LIN {X 0,Y 520.02,Z 1005.962,A -85,B 0,C 180,E1 24758.515,E2 24758.515} C_VEL
LIN {X 0,Y 519.949,Z 1010.979,A -85,B 0,C 180,E1 24756.515,E2 24756.515} C_VEL
LIN {X 0,Y 519.92,Z 1015.106,A -85,B 0,C 180,E1 24754.191,E2 24754.191} C_VEL
LIN {X 0,Y 519.914,Z 1017.318,A -85,B 0,C 180,E1 24751.984,E2 24751.984} C_VEL
LIN {X 0,Y 519.902,Z 1017.94,A -85,B 0,C 180,E1 24749.67,E2 24749.67} C_VEL
LIN {X 0,Y 519.907,Z 1016.99,A -85,B 0,C 180,E1 24747.576,E2 24747.576} C_VEL
LIN {X 0,Y 519.922,Z 1014.322,A -85,B 0,C 180,E1 24745.257,E2 24745.257} C_VEL
LIN {X 0,Y 519.954,Z 1010.226,A -85,B 0,C 180,E1 24743.153,E2 24743.153} C_VEL
LIN {X 0,Y 520.031,Z 1004.711,A -85,B 0,C 180,E1 24741.041,E2 24741.041} C_VEL
LIN {X 0,Y 520.195,Z 996.956,A -85,B 0,C 180,E1 24738.807,E2 24738.807} C_VEL
LIN {X 0,Y 520.466,Z 988.312,A -85,B 0,C 180,E1 24736.785,E2 24736.785} C_VEL
LIN {X 0,Y 520.856,Z 977.732,A -85,B 0,C 180,E1 24734.753,E2 24734.753} C_VEL
LIN {X 0,Y 521.388,Z 965.862,A -85,B 0,C 180,E1 24732.824,E2 24732.824} C_VEL
LIN {X 0,Y 522.046,Z 952.484,A -85,B 0,C 180,E1 24730.999,E2 24730.999} C_VEL
LIN {X 0,Y 522.795,Z 938.835,A -85,B 0,C 180,E1 24729.397,E2 24729.397} C_VEL
LIN {X 0,Y 523.77,Z 921.534,A -85,B 0,C 180,E1 24727.674,E2 24727.674} C_VEL
LIN {X 0,Y 524.742,Z 904.295,A -85,B 0,C 180,E1 24726.235,E2 24726.235} C_VEL
LIN {X 0,Y 525.694,Z 885.972,A -85,B 0,C 180,E1 24724.964,E2 24724.964} C_VEL
LIN {X 0,Y 526.661,Z 866.688,A -85,B 0,C 180,E1 24723.868,E2 24723.868} C_VEL
LIN {X 0,Y 527.517,Z 847.072,A -85,B 0,C 180,E1 24722.979,E2 24722.979} C_VEL
LIN {X 0,Y 528.202,Z 826.709,A -85,B 0,C 180,E1 24722.278,E2 24722.278} C_VEL
LIN {X 0,Y 528.779,Z 805.763,A -85,B 0,C 180,E1 24721.772,E2 24721.772} C_VEL
LIN {X 0,Y 529.175,Z 772.046,A -85,B 0,C 180,E1 24721.252,E2 24721.252} C_VEL
LIN {X 0,Y 534.131,Z 754.98,A -85,B 0,C 180,E1 24720.384,E2 24720.384} C_VEL
LIN {X 0,Y 537.725,Z 746.024,A -85,B 0,C 180,E1 24719.988,E2 24719.988} C_VEL
LIN {X 0,Y 541.751,Z 735.129,A -85,B 0,C 180,E1 24719.5,E2 24719.5} C_VEL
LIN {X 0,Y 548.246,Z 721.737,A -85,B 0,C 180,E1 24719.05,E2 24719.05} C_VEL
LIN {X 0,Y 556.194,Z 706.531,A -85,B 0,C 180,E1 24718.739,E2 24718.739} C_VEL
LIN {X 0,Y 561.276,Z 695.809,A -85,B 0,C 180,E1 24718.597,E2 24718.597} C_VEL
LIN {X 0,Y 565.411,Z 684.381,A -85,B 0,C 180,E1 24718.275,E2 24718.275} C_VEL
LIN {X 0,Y 572.184,Z 665.163,A -85,B 0,C 180,E1 24717.972,E2 24717.972} C_VEL
LIN {X 0,Y 577.855,Z 644.455,A -85,B 0,C 180,E1 24717.756,E2 24717.756} C_VEL
LIN {X 0,Y 581.468,Z 624.036,A -85,B 0,C 180,E1 24717.559,E2 24717.559} C_VEL
LIN {X 0,Y 581.827,Z 621.745,A -85,B 0,C 180,E1 24717.519,E2 24717.519} C_VEL
LIN {X 0,Y 583.33,Z 625.442,A -85,B 0,C 180,E1 24716.971,E2 24716.971} C_VEL
LIN {X 0,Y 583.255,Z 628.304,A -85,B 0,C 180,E1 24716.379,E2 24716.379} C_VEL
LIN {X 0,Y 581.69,Z 630.179,A -85,B 0,C 180,E1 24715.769,E2 24715.769} C_VEL
LIN {X 0,Y 578.618,Z 631.026,A -85,B 0,C 180,E1 24715.165,E2 24715.165} C_VEL
LIN {X 0,Y 574.8,Z 630.645,A -85,B 0,C 180,E1 24714.668,E2 24714.668} C_VEL
LIN {X 0,Y 568.857,Z 628.613,A -85,B 0,C 180,E1 24714.123,E2 24714.123} C_VEL
LIN {X 0,Y 560.136,Z 623.948,A -85,B 0,C 180,E1 24713.271,E2 24713.271} C_VEL
LIN {X 0,Y 552.133,Z 617.574,A -85,B 0,C 180,E1 24712.313,E2 24712.313} C_VEL
LIN {X 0,Y 545.581,Z 609.876,A -85,B 0,C 180,E1 24711.323,E2 24711.323} C_VEL
LIN {X 0,Y 540.263,Z 600.41,A -85,B 0,C 180,E1 24710.26,E2 24710.26} C_VEL
LIN {X 0,Y 536.466,Z 589.095,A -85,B 0,C 180,E1 24709.143,E2 24709.143} C_VEL
LIN {X 0,Y 534.195,Z 576.156,A -85,B 0,C 180,E1 24707.993,E2 24707.993} C_VEL
LIN {X 0,Y 533.452,Z 558.89,A -85,B 0,C 180,E1 24706.613,E2 24706.613} C_VEL
LIN {X 0,Y 535.809,Z 510.668,A -85,B 0,C 180,E1 24702.989,E2 24702.989} C_VEL
LIN {X 0,Y 537.167,Z 485.07,A -85,B 0,C 180,E1 24701.005,E2 24701.005} C_VEL
LIN {X 0,Y 528.374,Z 467.062,A -85,B 0,C 180,E1 24698.504,E2 24698.504} C_VEL
LIN {X 0,Y 523.968,Z 458.341,A -85,B 0,C 180,E1 24697.222,E2 24697.222} C_VEL
LIN {X 0,Y 521.991,Z 454.315,A -85,B 0,C 180,E1 24696.624,E2 24696.624} C_VEL
LIN {X 0,Y 520.59,Z 450.764,A -85,B 0,C 180,E1 24696.131,E2 24696.131} C_VEL
LIN {X 0,Y 520.581,Z 450.636,A -85,B 0,C 180,E1 24692.729,E2 24692.729} C_VEL
LIN {X 0,Y 520.553,Z 450.643,A -85,B 0,C 180,E1 24689.306,E2 24689.306} C_VEL
LIN {X 0,Y 520.585,Z 450.64,A -85,B 0,C 180,E1 24685.848,E2 24685.848} C_VEL
LIN {X 0,Y 520.561,Z 450.642,A -85,B 0,C 180,E1 24682.471,E2 24682.471} C_VEL
LIN {X 0,Y 520.537,Z 450.644,A -85,B 0,C 180,E1 24678.942,E2 24678.942} C_VEL
LIN {X 0,Y 520.586,Z 450.638,A -85,B 0,C 180,E1 24675.598,E2 24675.598} C_VEL
LIN {X 0,Y 520.533,Z 450.645,A -85,B 0,C 180,E1 24672.198,E2 24672.198} C_VEL
LIN {X 0,Y 520.562,Z 450.641,A -85,B 0,C 180,E1 24668.616,E2 24668.616} C_VEL
LIN {X 0,Y 520.585,Z 450.639,A -85,B 0,C 180,E1 24665.179,E2 24665.179} C_VEL
LIN {X 0,Y 520.563,Z 450.644,A -85,B 0,C 180,E1 24661.651,E2 24661.651} C_VEL
LIN {X 0,Y 520.583,Z 450.641,A -85,B 0,C 180,E1 24658.239,E2 24658.239} C_VEL
LIN {X 0,Y 520.573,Z 450.644,A -85,B 0,C 180,E1 24654.821,E2 24654.821} C_VEL
LIN {X 0,Y 520.584,Z 450.635,A -85,B 0,C 180,E1 24651.384,E2 24651.384} C_VEL
LIN {X 0,Y 520.559,Z 450.637,A -85,B 0,C 180,E1 24647.915,E2 24647.915} C_VEL
LIN {X 0,Y 520.582,Z 450.639,A -85,B 0,C 180,E1 24644.401,E2 24644.401} C_VEL
LIN {X 0,Y 520.565,Z 450.638,A -85,B 0,C 180,E1 24640.942,E2 24640.942} C_VEL
LIN {X 0,Y 520.533,Z 450.636,A -85,B 0,C 180,E1 24637.408,E2 24637.408} C_VEL
LIN {X 0,Y 520.584,Z 450.636,A -85,B 0,C 180,E1 24634.008,E2 24634.008} C_VEL
LIN {X 0,Y 520.541,Z 450.644,A -85,B 0,C 180,E1 24630.672,E2 24630.672} C_VEL
LIN {X 0,Y 520.557,Z 450.643,A -85,B 0,C 180,E1 24627.204,E2 24627.204} C_VEL
LIN {X 0,Y 520.586,Z 450.639,A -85,B 0,C 180,E1 24623.732,E2 24623.732} C_VEL
LIN {X 0,Y 520.556,Z 450.645,A -85,B 0,C 180,E1 24620.237,E2 24620.237} C_VEL
LIN {X 0,Y 520.586,Z 450.64,A -85,B 0,C 180,E1 24617.852,E2 24617.852} C_VEL
LIN {X 0,Y 519.595,Z 450.764,A -85,B 0,C 180,E1 24617.004,E2 24617.004} C_VEL
LIN {X 0,Y 513.124,Z 451.571,A -85,B 0,C 180,E1 24614.622,E2 24614.622} C_VEL
LIN {X 0,Y 512.608,Z 451.631,A -85,B 0,C 180,E1 24614.001,E2 24614.001} C_VEL
LIN {X 0,Y 512.622,Z 451.634,A -85,B 0,C 180,E1 24610.475,E2 24610.475} C_VEL
LIN {X 0,Y 512.655,Z 451.706,A -85,B 0,C 180,E1 24607.253,E2 24607.253} C_VEL
LIN {X 0,Y 522.069,Z 477.016,A -85,B 0,C 180,E1 24604.288,E2 24604.288} C_VEL
LIN {X 0,Y 521.564,Z 496.747,A -85,B 0,C 180,E1 24602.718,E2 24602.718} C_VEL
LIN {X 0,Y 524.472,Z 512.948,A -85,B 0,C 180,E1 24602.253,E2 24602.253} C_VEL
LIN {X 0,Y 521.733,Z 755.843,A -85,B 0,C 180,E1 24598.599,E2 24598.599} C_VEL
LIN {X 0,Y 521.118,Z 776.945,A -85,B 0,C 180,E1 24598.086,E2 24598.086} C_VEL
LIN {X 0,Y 520.343,Z 797.387,A -85,B 0,C 180,E1 24597.369,E2 24597.369} C_VEL
LIN {X 0,Y 519.455,Z 815.917,A -85,B 0,C 180,E1 24596.522,E2 24596.522} C_VEL
LIN {X 0,Y 518.399,Z 835.331,A -85,B 0,C 180,E1 24595.413,E2 24595.413} C_VEL
LIN {X 0,Y 517.335,Z 853.73,A -85,B 0,C 180,E1 24594.127,E2 24594.127} C_VEL
LIN {X 0,Y 516.225,Z 871.52,A -85,B 0,C 180,E1 24592.628,E2 24592.628} C_VEL
LIN {X 0,Y 515.211,Z 887.582,A -85,B 0,C 180,E1 24591.018,E2 24591.018} C_VEL
LIN {X 0,Y 514.336,Z 902.16,A -85,B 0,C 180,E1 24589.297,E2 24589.297} C_VEL
LIN {X 0,Y 513.544,Z 916.286,A -85,B 0,C 180,E1 24587.33,E2 24587.33} C_VEL
LIN {X 0,Y 512.924,Z 928.972,A -85,B 0,C 180,E1 24585.221,E2 24585.221} C_VEL
LIN {X 0,Y 512.488,Z 939.658,A -85,B 0,C 180,E1 24583.08,E2 24583.08} C_VEL
LIN {X 0,Y 512.196,Z 948.513,A -85,B 0,C 180,E1 24580.914,E2 24580.914} C_VEL
LIN {X 0,Y 512.04,Z 955.576,A -85,B 0,C 180,E1 24578.76,E2 24578.76} C_VEL
LIN {X 0,Y 511.954,Z 961.153,A -85,B 0,C 180,E1 24576.504,E2 24576.504} C_VEL
LIN {X 0,Y 511.921,Z 965.02,A -85,B 0,C 180,E1 24574.256,E2 24574.256} C_VEL
LIN {X 0,Y 511.912,Z 967.346,A -85,B 0,C 180,E1 24571.902,E2 24571.902} C_VEL
LIN {X 0,Y 511.903,Z 967.949,A -85,B 0,C 180,E1 24569.664,E2 24569.664} C_VEL
LIN {X 0,Y 511.906,Z 966.99,A -85,B 0,C 180,E1 24567.425,E2 24567.425} C_VEL
LIN {X 0,Y 511.924,Z 964.355,A -85,B 0,C 180,E1 24565.182,E2 24565.182} C_VEL
LIN {X 0,Y 511.958,Z 960.09,A -85,B 0,C 180,E1 24562.932,E2 24562.932} C_VEL
LIN {X 0,Y 512.054,Z 954.108,A -85,B 0,C 180,E1 24560.672,E2 24560.672} C_VEL
LIN {X 0,Y 512.254,Z 946.567,A -85,B 0,C 180,E1 24558.478,E2 24558.478} C_VEL
LIN {X 0,Y 512.578,Z 937.474,A -85,B 0,C 180,E1 24556.347,E2 24556.347} C_VEL
LIN {X 0,Y 513.066,Z 926.091,A -85,B 0,C 180,E1 24554.167,E2 24554.167} C_VEL
LIN {X 0,Y 513.736,Z 913.04,A -85,B 0,C 180,E1 24552.09,E2 24552.09} C_VEL
LIN {X 0,Y 514.521,Z 899.191,A -85,B 0,C 180,E1 24550.236,E2 24550.236} C_VEL
LIN {X 0,Y 515.417,Z 884.365,A -85,B 0,C 180,E1 24548.55,E2 24548.55} C_VEL
LIN {X 0,Y 516.418,Z 868.089,A -85,B 0,C 180,E1 24546.976,E2 24546.976} C_VEL
LIN {X 0,Y 517.483,Z 850.915,A -85,B 0,C 180,E1 24545.576,E2 24545.576} C_VEL
LIN {X 0,Y 518.537,Z 832.917,A -85,B 0,C 180,E1 24544.348,E2 24544.348} C_VEL
LIN {X 0,Y 519.552,Z 814.203,A -85,B 0,C 180,E1 24543.297,E2 24543.297} C_VEL
LIN {X 0,Y 520.482,Z 794.444,A -85,B 0,C 180,E1 24542.421,E2 24542.421} C_VEL
LIN {X 0,Y 521.208,Z 774.575,A -85,B 0,C 180,E1 24541.755,E2 24541.755} C_VEL
LIN {X 0,Y 521.766,Z 754.007,A -85,B 0,C 180,E1 24541.277,E2 24541.277} C_VEL
LIN {X 0,Y 524.313,Z 517.721,A -85,B 0,C 180,E1 24537.722,E2 24537.722} C_VEL
LIN {X 0,Y 519.038,Z 498.46,A -85,B 0,C 180,E1 24537.028,E2 24537.028} C_VEL
LIN {X 0,Y 519.95,Z 475.219,A -85,B 0,C 180,E1 24534.157,E2 24534.157} C_VEL
LIN {X 0,Y 514.832,Z 458.731,A -85,B 0,C 180,E1 24531.575,E2 24531.575} C_VEL
LIN {X 0,Y 512.627,Z 451.637,A -85,B 0,C 180,E1 24530.417,E2 24530.417} C_VEL
LIN {X 0,Y 512.646,Z 451.628,A -85,B 0,C 180,E1 24526.949,E2 24526.949} C_VEL
LIN {X 0,Y 512.633,Z 451.628,A -85,B 0,C 180,E1 24523.483,E2 24523.483} C_VEL
LIN {X 0,Y 512.63,Z 451.628,A -85,B 0,C 180,E1 24519.919,E2 24519.919} C_VEL
LIN {X 0,Y 512.638,Z 451.63,A -85,B 0,C 180,E1 24516.504,E2 24516.504} C_VEL
LIN {X 0,Y 512.638,Z 451.637,A -85,B 0,C 180,E1 24512.968,E2 24512.968} C_VEL
LIN {X 0,Y 512.667,Z 451.773,A -85,B 0,C 180,E1 24512.038,E2 24512.038} C_VEL
LIN {X 0,Y 520.423,Z 474.252,A -85,B 0,C 180,E1 24509.053,E2 24509.053} C_VEL
LIN {X 0,Y 521.005,Z 476.298,A -85,B 0,C 180,E1 24508.796,E2 24508.796} C_VEL
LIN {X 0,Y 519.755,Z 507.875,A -85,B 0,C 180,E1 24505.648,E2 24505.648} C_VEL
LIN {X 0,Y 518.449,Z 542.34,A -85,B 0,C 180,E1 24502.269,E2 24502.269} C_VEL
LIN {X 0,Y 517.128,Z 577.872,A -85,B 0,C 180,E1 24498.838,E2 24498.838} C_VEL
LIN {X 0,Y 516.275,Z 609.248,A -85,B 0,C 180,E1 24495.884,E2 24495.884} C_VEL
LIN {X 0,Y 516.883,Z 614.725,A -85,B 0,C 180,E1 24495.767,E2 24495.767} C_VEL
LIN {X 0,Y 515.399,Z 751.101,A -85,B 0,C 180,E1 24493.597,E2 24493.597} C_VEL
LIN {X 0,Y 515.196,Z 767.868,A -85,B 0,C 180,E1 24493.11,E2 24493.11} C_VEL
LIN {X 0,Y 514.884,Z 783.198,A -85,B 0,C 180,E1 24492.448,E2 24492.448} C_VEL
LIN {X 0,Y 514.483,Z 798.649,A -85,B 0,C 180,E1 24491.547,E2 24491.547} C_VEL
LIN {X 0,Y 514.057,Z 812.03,A -85,B 0,C 180,E1 24490.535,E2 24490.535} C_VEL
LIN {X 0,Y 513.602,Z 825.042,A -85,B 0,C 180,E1 24489.299,E2 24489.299} C_VEL
LIN {X 0,Y 513.201,Z 836.355,A -85,B 0,C 180,E1 24487.951,E2 24487.951} C_VEL
LIN {X 0,Y 512.843,Z 846.858,A -85,B 0,C 180,E1 24486.381,E2 24486.381} C_VEL
LIN {X 0,Y 512.595,Z 855.085,A -85,B 0,C 180,E1 24484.812,E2 24484.812} C_VEL
LIN {X 0,Y 512.416,Z 861.858,A -85,B 0,C 180,E1 24483.132,E2 24483.132} C_VEL
LIN {X 0,Y 512.306,Z 866.86,A -85,B 0,C 180,E1 24481.454,E2 24481.454} C_VEL
LIN {X 0,Y 512.257,Z 870.497,A -85,B 0,C 180,E1 24479.553,E2 24479.553} C_VEL
LIN {X 0,Y 512.241,Z 872.22,A -85,B 0,C 180,E1 24477.763,E2 24477.763} C_VEL
LIN {X 0,Y 512.262,Z 872.167,A -85,B 0,C 180,E1 24475.859,E2 24475.859} C_VEL
LIN {X 0,Y 512.314,Z 870.441,A -85,B 0,C 180,E1 24474.063,E2 24474.063} C_VEL
LIN {X 0,Y 512.407,Z 866.934,A -85,B 0,C 180,E1 24472.262,E2 24472.262} C_VEL
LIN {X 0,Y 512.594,Z 861.578,A -85,B 0,C 180,E1 24470.456,E2 24470.456} C_VEL
LIN {X 0,Y 512.822,Z 854.415,A -85,B 0,C 180,E1 24468.731,E2 24468.731} C_VEL
LIN {X 0,Y 513.149,Z 846.02,A -85,B 0,C 180,E1 24467.166,E2 24467.166} C_VEL
LIN {X 0,Y 513.505,Z 836.727,A -85,B 0,C 180,E1 24465.798,E2 24465.798} C_VEL
LIN {X 0,Y 513.961,Z 825.126,A -85,B 0,C 180,E1 24464.427,E2 24464.427} C_VEL
LIN {X 0,Y 514.405,Z 812.983,A -85,B 0,C 180,E1 24463.282,E2 24463.282} C_VEL
LIN {X 0,Y 514.82,Z 799.097,A -85,B 0,C 180,E1 24462.247,E2 24462.247} C_VEL
LIN {X 0,Y 515.154,Z 785.148,A -85,B 0,C 180,E1 24461.44,E2 24461.44} C_VEL
LIN {X 0,Y 515.389,Z 769.335,A -85,B 0,C 180,E1 24460.773,E2 24460.773} C_VEL
LIN {X 0,Y 515.494,Z 753.566,A -85,B 0,C 180,E1 24460.325,E2 24460.325} C_VEL
LIN {X 0,Y 517.063,Z 653.13,A -85,B 0,C 180,E1 24458.571,E2 24458.571} C_VEL
LIN {X 0,Y 517.869,Z 619.502,A -85,B 0,C 180,E1 24457.943,E2 24457.943} C_VEL
LIN {X 0,Y 519.364,Z 614.58,A -85,B 0,C 180,E1 24457.531,E2 24457.531} C_VEL
LIN {X 0,Y 522.354,Z 579.387,A -85,B 0,C 180,E1 24453.758,E2 24453.758} C_VEL
LIN {X 0,Y 526.373,Z 547.133,A -85,B 0,C 180,E1 24450.091,E2 24450.091} C_VEL
LIN {X 0,Y 530.894,Z 521.985,A -85,B 0,C 180,E1 24447.024,E2 24447.024} C_VEL
LIN {X 0,Y 534.242,Z 508.14,A -85,B 0,C 180,E1 24445.193,E2 24445.193} C_VEL
LIN {X 0,Y 536.725,Z 498.815,A -85,B 0,C 180,E1 24443.769,E2 24443.769} C_VEL
LIN {X 0,Y 536.061,Z 495.319,A -85,B 0,C 180,E1 24442.417,E2 24442.417} C_VEL
LIN {X 0,Y 536.022,Z 493.334,A -85,B 0,C 180,E1 24441.189,E2 24441.189} C_VEL
LIN {X 0,Y 536.329,Z 493.269,A -85,B 0,C 180,E1 24439.832,E2 24439.832} C_VEL
LIN {X 0,Y 536.826,Z 494.261,A -85,B 0,C 180,E1 24439.049,E2 24439.049} C_VEL
LIN {X 0,Y 531.613,Z 507.135,A -85,B 0,C 180,E1 24437.66,E2 24437.66} C_VEL
LIN {X 0,Y 527.47,Z 522.779,A -85,B 0,C 180,E1 24436.16,E2 24436.16} C_VEL
LIN {X 0,Y 523.936,Z 544.359,A -85,B 0,C 180,E1 24434.304,E2 24434.304} C_VEL
LIN {X 0,Y 522.918,Z 563.007,A -85,B 0,C 180,E1 24432.75,E2 24432.75} C_VEL
LIN {X 0,Y 523.903,Z 578.013,A -85,B 0,C 180,E1 24431.472,E2 24431.472} C_VEL
LIN {X 0,Y 526.805,Z 591.429,A -85,B 0,C 180,E1 24430.272,E2 24430.272} C_VEL
LIN {X 0,Y 531.066,Z 602.392,A -85,B 0,C 180,E1 24429.243,E2 24429.243} C_VEL
LIN {X 0,Y 537.171,Z 612.519,A -85,B 0,C 180,E1 24428.235,E2 24428.235} C_VEL
LIN {X 0,Y 544.544,Z 621.028,A -85,B 0,C 180,E1 24427.341,E2 24427.341} C_VEL
LIN {X 0,Y 553.465,Z 628.474,A -85,B 0,C 180,E1 24426.495,E2 24426.495} C_VEL
LIN {X 0,Y 563.066,Z 634.265,A -85,B 0,C 180,E1 24425.756,E2 24425.756} C_VEL
LIN {X 0,Y 569.587,Z 637.069,A -85,B 0,C 180,E1 24425.288,E2 24425.288} C_VEL
LIN {X 0,Y 573.909,Z 638.04,A -85,B 0,C 180,E1 24424.851,E2 24424.851} C_VEL
LIN {X 0,Y 577.534,Z 637.952,A -85,B 0,C 180,E1 24424.33,E2 24424.33} C_VEL
LIN {X 0,Y 580.243,Z 636.66,A -85,B 0,C 180,E1 24423.702,E2 24423.702} C_VEL
LIN {X 0,Y 581.263,Z 634.732,A -85,B 0,C 180,E1 24423.118,E2 24423.118} C_VEL
LIN {X 0,Y 574.611,Z 654.779,A -85,B 0,C 180,E1 24422.941,E2 24422.941} C_VEL
LIN {X 0,Y 566.188,Z 674.796,A -85,B 0,C 180,E1 24422.656,E2 24422.656} C_VEL
LIN {X 0,Y 558.971,Z 690.695,A -85,B 0,C 180,E1 24422.273,E2 24422.273} C_VEL
LIN {X 0,Y 556.522,Z 696.659,A -85,B 0,C 180,E1 24422.067,E2 24422.067} C_VEL
LIN {X 0,Y 546.748,Z 712.537,A -85,B 0,C 180,E1 24421.714,E2 24421.714} C_VEL
LIN {X 0,Y 538.402,Z 726.619,A -85,B 0,C 180,E1 24421.207,E2 24421.207} C_VEL
LIN {X 0,Y 532.513,Z 739.169,A -85,B 0,C 180,E1 24420.65,E2 24420.65} C_VEL
LIN {X 0,Y 529.342,Z 747.906,A -85,B 0,C 180,E1 24420.225,E2 24420.225} C_VEL
LIN {X 0,Y 525.03,Z 759.145,A -85,B 0,C 180,E1 24419.68,E2 24419.68} C_VEL
LIN {X 0,Y 521.684,Z 771.68,A -85,B 0,C 180,E1 24419.052,E2 24419.052} C_VEL
LIN {X 0,Y 521.265,Z 808.1,A -85,B 0,C 180,E1 24418.499,E2 24418.499} C_VEL
LIN {X 0,Y 520.716,Z 830.208,A -85,B 0,C 180,E1 24417.958,E2 24417.958} C_VEL
LIN {X 0,Y 520.042,Z 850.995,A -85,B 0,C 180,E1 24417.232,E2 24417.232} C_VEL
LIN {X 0,Y 519.241,Z 869.965,A -85,B 0,C 180,E1 24416.351,E2 24416.351} C_VEL
LIN {X 0,Y 518.204,Z 888.718,A -85,B 0,C 180,E1 24415.241,E2 24415.241} C_VEL
LIN {X 0,Y 517.097,Z 907.27,A -85,B 0,C 180,E1 24413.891,E2 24413.891} C_VEL
LIN {X 0,Y 516.031,Z 924.658,A -85,B 0,C 180,E1 24412.38,E2 24412.38} C_VEL
LIN {X 0,Y 515.042,Z 940.356,A -85,B 0,C 180,E1 24410.751,E2 24410.751} C_VEL
LIN {X 0,Y 514.26,Z 953.384,A -85,B 0,C 180,E1 24409.183,E2 24409.183} C_VEL
LIN {X 0,Y 513.49,Z 967.318,A -85,B 0,C 180,E1 24407.216,E2 24407.216} C_VEL
LIN {X 0,Y 512.95,Z 978.366,A -85,B 0,C 180,E1 24405.373,E2 24405.373} C_VEL
LIN {X 0,Y 512.48,Z 989.843,A -85,B 0,C 180,E1 24403.081,E2 24403.081} C_VEL
LIN {X 0,Y 512.191,Z 998.694,A -85,B 0,C 180,E1 24400.914,E2 24400.914} C_VEL
LIN {X 0,Y 512.033,Z 1005.958,A -85,B 0,C 180,E1 24398.648,E2 24398.648} C_VEL
LIN {X 0,Y 511.955,Z 1010.977,A -85,B 0,C 180,E1 24396.617,E2 24396.617} C_VEL
LIN {X 0,Y 511.919,Z 1015.101,A -85,B 0,C 180,E1 24394.257,E2 24394.257} C_VEL
LIN {X 0,Y 511.914,Z 1017.314,A -85,B 0,C 180,E1 24392.015,E2 24392.015} C_VEL
LIN {X 0,Y 511.902,Z 1017.94,A -85,B 0,C 180,E1 24389.665,E2 24389.665} C_VEL
LIN {X 0,Y 511.907,Z 1016.985,A -85,B 0,C 180,E1 24387.538,E2 24387.538} C_VEL
LIN {X 0,Y 511.923,Z 1014.322,A -85,B 0,C 180,E1 24385.183,E2 24385.183} C_VEL
LIN {X 0,Y 511.957,Z 1010.224,A -85,B 0,C 180,E1 24383.046,E2 24383.046} C_VEL
LIN {X 0,Y 512.045,Z 1004.71,A -85,B 0,C 180,E1 24380.9,E2 24380.9} C_VEL
LIN {X 0,Y 512.223,Z 997.388,A -85,B 0,C 180,E1 24378.744,E2 24378.744} C_VEL
LIN {X 0,Y 512.519,Z 988.832,A -85,B 0,C 180,E1 24376.692,E2 24376.692} C_VEL
LIN {X 0,Y 512.979,Z 977.728,A -85,B 0,C 180,E1 24374.513,E2 24374.513} C_VEL
LIN {X 0,Y 513.58,Z 965.794,A -85,B 0,C 180,E1 24372.544,E2 24372.544} C_VEL
LIN {X 0,Y 514.31,Z 952.479,A -85,B 0,C 180,E1 24370.702,E2 24370.702} C_VEL
LIN {X 0,Y 515.136,Z 938.829,A -85,B 0,C 180,E1 24369.076,E2 24369.076} C_VEL
LIN {X 0,Y 516.22,Z 921.531,A -85,B 0,C 180,E1 24367.33,E2 24367.33} C_VEL
LIN {X 0,Y 517.306,Z 904.221,A -85,B 0,C 180,E1 24365.866,E2 24365.866} C_VEL
LIN {X 0,Y 518.352,Z 885.967,A -85,B 0,C 180,E1 24364.585,E2 24364.585} C_VEL
LIN {X 0,Y 519.339,Z 867.859,A -85,B 0,C 180,E1 24363.539,E2 24363.539} C_VEL
LIN {X 0,Y 520.181,Z 848.295,A -85,B 0,C 180,E1 24362.653,E2 24362.653} C_VEL
LIN {X 0,Y 520.884,Z 827.337,A -85,B 0,C 180,E1 24361.932,E2 24361.932} C_VEL
LIN {X 0,Y 521.509,Z 805.279,A -85,B 0,C 180,E1 24361.398,E2 24361.398} C_VEL
LIN {X 0,Y 522.015,Z 771.041,A -85,B 0,C 180,E1 24360.861,E2 24360.861} C_VEL
LIN {X 0,Y 527.015,Z 754.196,A -85,B 0,C 180,E1 24359.998,E2 24359.998} C_VEL
LIN {X 0,Y 530.862,Z 744.608,A -85,B 0,C 180,E1 24359.56,E2 24359.56} C_VEL
LIN {X 0,Y 535.34,Z 733.098,A -85,B 0,C 180,E1 24359.033,E2 24359.033} C_VEL
LIN {X 0,Y 542.601,Z 719.324,A -85,B 0,C 180,E1 24358.507,E2 24358.507} C_VEL
LIN {X 0,Y 552.028,Z 704.082,A -85,B 0,C 180,E1 24358.071,E2 24358.071} C_VEL
LIN {X 0,Y 556.94,Z 695.681,A -85,B 0,C 180,E1 24357.901,E2 24357.901} C_VEL
LIN {X 0,Y 562.319,Z 683.23,A -85,B 0,C 180,E1 24357.522,E2 24357.522} C_VEL
LIN {X 0,Y 570.851,Z 664.161,A -85,B 0,C 180,E1 24357.174,E2 24357.174} C_VEL
LIN {X 0,Y 578.175,Z 644.792,A -85,B 0,C 180,E1 24356.963,E2 24356.963} C_VEL
LIN {X 0,Y 581.311,Z 634.577,A -85,B 0,C 180,E1 24356.871,E2 24356.871} C_VEL
LIN {X 0,Y 580.248,Z 636.656,A -85,B 0,C 180,E1 24356.3,E2 24356.3} C_VEL
LIN {X 0,Y 578.071,Z 637.821,A -85,B 0,C 180,E1 24355.768,E2 24355.768} C_VEL
LIN {X 0,Y 574.538,Z 638.101,A -85,B 0,C 180,E1 24355.226,E2 24355.226} C_VEL
LIN {X 0,Y 570.275,Z 637.279,A -85,B 0,C 180,E1 24354.773,E2 24354.773} C_VEL
LIN {X 0,Y 560.456,Z 633.212,A -85,B 0,C 180,E1 24353.916,E2 24353.916} C_VEL
LIN {X 0,Y 551.304,Z 627.408,A -85,B 0,C 180,E1 24352.939,E2 24352.939} C_VEL
LIN {X 0,Y 543.628,Z 620.254,A -85,B 0,C 180,E1 24351.924,E2 24351.924} C_VEL
LIN {X 0,Y 537.412,Z 611.822,A -85,B 0,C 180,E1 24350.88,E2 24350.88} C_VEL
LIN {X 0,Y 532.658,Z 602.127,A -85,B 0,C 180,E1 24349.816,E2 24349.816} C_VEL
LIN {X 0,Y 529.071,Z 589.803,A -85,B 0,C 180,E1 24348.613,E2 24348.613} C_VEL
LIN {X 0,Y 527.134,Z 575.752,A -85,B 0,C 180,E1 24347.379,E2 24347.379} C_VEL
LIN {X 0,Y 526.882,Z 556.312,A -85,B 0,C 180,E1 24345.834,E2 24345.834} C_VEL
LIN {X 0,Y 529.293,Z 514.033,A -85,B 0,C 180,E1 24342.627,E2 24342.627} C_VEL
LIN {X 0,Y 530.745,Z 489.136,A -85,B 0,C 180,E1 24340.679,E2 24340.679} C_VEL
LIN {X 0,Y 522.147,Z 471.547,A -85,B 0,C 180,E1 24338.207,E2 24338.207} C_VEL
LIN {X 0,Y 515.983,Z 459.211,A -85,B 0,C 180,E1 24336.367,E2 24336.367} C_VEL
LIN {X 0,Y 514.262,Z 455.59,A -85,B 0,C 180,E1 24335.818,E2 24335.818} C_VEL
LIN {X 0,Y 512.684,Z 452.156,A -85,B 0,C 180,E1 24335.3,E2 24335.3} C_VEL
LIN {X 0,Y 512.605,Z 451.631,A -85,B 0,C 180,E1 24335.188,E2 24335.188} C_VEL
LIN {X 0,Y 512.644,Z 451.621,A -85,B 0,C 180,E1 24331.645,E2 24331.645} C_VEL
LIN {X 0,Y 512.617,Z 451.632,A -85,B 0,C 180,E1 24328.292,E2 24328.292} C_VEL
LIN {X 0,Y 512.641,Z 451.631,A -85,B 0,C 180,E1 24324.793,E2 24324.793} C_VEL
LIN {X 0,Y 512.639,Z 451.631,A -85,B 0,C 180,E1 24321.271,E2 24321.271} C_VEL
LIN {X 0,Y 512.651,Z 451.629,A -85,B 0,C 180,E1 24317.713,E2 24317.713} C_VEL
LIN {X 0,Y 512.622,Z 451.632,A -85,B 0,C 180,E1 24314.216,E2 24314.216} C_VEL
LIN {X 0,Y 512.597,Z 451.634,A -85,B 0,C 180,E1 24310.679,E2 24310.679} C_VEL
LIN {X 0,Y 512.651,Z 451.625,A -85,B 0,C 180,E1 24307.283,E2 24307.283} C_VEL
LIN {X 0,Y 512.594,Z 451.634,A -85,B 0,C 180,E1 24303.914,E2 24303.914} C_VEL
LIN {X 0,Y 512.622,Z 451.628,A -85,B 0,C 180,E1 24300.335,E2 24300.335} C_VEL
LIN {X 0,Y 512.645,Z 451.628,A -85,B 0,C 180,E1 24296.869,E2 24296.869} C_VEL
LIN {X 0,Y 512.631,Z 451.628,A -85,B 0,C 180,E1 24293.279,E2 24293.279} C_VEL
LIN {X 0,Y 512.641,Z 451.632,A -85,B 0,C 180,E1 24289.776,E2 24289.776} C_VEL
LIN {X 0,Y 512.627,Z 451.625,A -85,B 0,C 180,E1 24286.349,E2 24286.349} C_VEL
LIN {X 0,Y 512.645,Z 451.623,A -85,B 0,C 180,E1 24282.989,E2 24282.989} C_VEL
LIN {X 0,Y 512.618,Z 451.632,A -85,B 0,C 180,E1 24279.565,E2 24279.565} C_VEL
LIN {X 0,Y 512.637,Z 451.628,A -85,B 0,C 180,E1 24276.066,E2 24276.066} C_VEL
LIN {X 0,Y 512.627,Z 451.626,A -85,B 0,C 180,E1 24272.719,E2 24272.719} C_VEL
LIN {X 0,Y 512.594,Z 451.627,A -85,B 0,C 180,E1 24269.12,E2 24269.12} C_VEL
LIN {X 0,Y 512.644,Z 451.624,A -85,B 0,C 180,E1 24265.69,E2 24265.69} C_VEL
LIN {X 0,Y 512.602,Z 451.63,A -85,B 0,C 180,E1 24262.365,E2 24262.365} C_VEL
LIN {X 0,Y 512.617,Z 451.626,A -85,B 0,C 180,E1 24258.841,E2 24258.841} C_VEL
LIN {X 0,Y 512.651,Z 451.629,A -85,B 0,C 180,E1 24255.388,E2 24255.388} C_VEL
LIN {X 0,Y 512.608,Z 451.631,A -85,B 0,C 180,E1 24254.001,E2 24254.001} C_VEL
LIN {X 0,Y 511.64,Z 451.759,A -85,B 0,C 180,E1 24253.14,E2 24253.14} C_VEL
LIN {X 0,Y 505.215,Z 452.557,A -85,B 0,C 180,E1 24250.719,E2 24250.719} C_VEL
LIN {X 0,Y 504.704,Z 452.617,A -85,B 0,C 180,E1 24250.088,E2 24250.088} C_VEL
LIN {X 0,Y 504.702,Z 452.709,A -85,B 0,C 180,E1 24247.835,E2 24247.835} C_VEL
LIN {X 0,Y 513.665,Z 476.547,A -85,B 0,C 180,E1 24244.966,E2 24244.966} C_VEL
LIN {X 0,Y 515.013,Z 480.366,A -85,B 0,C 180,E1 24244.533,E2 24244.533} C_VEL
LIN {X 0,Y 514.614,Z 497.14,A -85,B 0,C 180,E1 24243.215,E2 24243.215} C_VEL
LIN {X 0,Y 517.714,Z 514.315,A -85,B 0,C 180,E1 24242.71,E2 24242.71} C_VEL
LIN {X 0,Y 514.722,Z 756.349,A -85,B 0,C 180,E1 24239.021,E2 24239.021} C_VEL
LIN {X 0,Y 514.073,Z 777.294,A -85,B 0,C 180,E1 24238.506,E2 24238.506} C_VEL
LIN {X 0,Y 513.25,Z 797.555,A -85,B 0,C 180,E1 24237.789,E2 24237.789} C_VEL
LIN {X 0,Y 512.279,Z 816.309,A -85,B 0,C 180,E1 24236.924,E2 24236.924} C_VEL
LIN {X 0,Y 511.192,Z 834.747,A -85,B 0,C 180,E1 24235.859,E2 24235.859} C_VEL
LIN {X 0,Y 509.955,Z 853.489,A -85,B 0,C 180,E1 24234.528,E2 24234.528} C_VEL
LIN {X 0,Y 508.683,Z 871.724,A -85,B 0,C 180,E1 24232.964,E2 24232.964} C_VEL
LIN {X 0,Y 507.598,Z 887.383,A -85,B 0,C 180,E1 24231.371,E2 24231.371} C_VEL
LIN {X 0,Y 506.619,Z 902.163,A -85,B 0,C 180,E1 24229.603,E2 24229.603} C_VEL
LIN {X 0,Y 505.742,Z 916.288,A -85,B 0,C 180,E1 24227.606,E2 24227.606} C_VEL
LIN {X 0,Y 505.059,Z 928.776,A -85,B 0,C 180,E1 24225.501,E2 24225.501} C_VEL
LIN {X 0,Y 504.573,Z 939.379,A -85,B 0,C 180,E1 24223.353,E2 24223.353} C_VEL
LIN {X 0,Y 504.245,Z 948.11,A -85,B 0,C 180,E1 24221.205,E2 24221.205} C_VEL
LIN {X 0,Y 504.051,Z 955.579,A -85,B 0,C 180,E1 24218.9,E2 24218.9} C_VEL
LIN {X 0,Y 503.959,Z 961.155,A -85,B 0,C 180,E1 24216.607,E2 24216.607} C_VEL
LIN {X 0,Y 503.921,Z 965.021,A -85,B 0,C 180,E1 24214.323,E2 24214.323} C_VEL
LIN {X 0,Y 503.913,Z 967.346,A -85,B 0,C 180,E1 24211.932,E2 24211.932} C_VEL
LIN {X 0,Y 503.904,Z 967.948,A -85,B 0,C 180,E1 24209.658,E2 24209.658} C_VEL
LIN {X 0,Y 503.906,Z 966.989,A -85,B 0,C 180,E1 24207.384,E2 24207.384} C_VEL
LIN {X 0,Y 503.924,Z 964.354,A -85,B 0,C 180,E1 24205.105,E2 24205.105} C_VEL
LIN {X 0,Y 503.962,Z 960.088,A -85,B 0,C 180,E1 24202.819,E2 24202.819} C_VEL
LIN {X 0,Y 504.076,Z 954.105,A -85,B 0,C 180,E1 24200.523,E2 24200.523} C_VEL
LIN {X 0,Y 504.296,Z 946.713,A -85,B 0,C 180,E1 24198.332,E2 24198.332} C_VEL
LIN {X 0,Y 504.656,Z 937.457,A -85,B 0,C 180,E1 24196.126,E2 24196.126} C_VEL
LIN {X 0,Y 505.207,Z 926.09,A -85,B 0,C 180,E1 24193.914,E2 24193.914} C_VEL
LIN {X 0,Y 505.948,Z 913.038,A -85,B 0,C 180,E1 24191.805,E2 24191.805} C_VEL
LIN {X 0,Y 506.841,Z 898.906,A -85,B 0,C 180,E1 24189.888,E2 24189.888} C_VEL
LIN {X 0,Y 507.851,Z 883.809,A -85,B 0,C 180,E1 24188.154,E2 24188.154} C_VEL
LIN {X 0,Y 508.977,Z 867.319,A -85,B 0,C 180,E1 24186.549,E2 24186.549} C_VEL
LIN {X 0,Y 510.204,Z 849.48,A -85,B 0,C 180,E1 24185.08,E2 24185.08} C_VEL
LIN {X 0,Y 511.414,Z 830.921,A -85,B 0,C 180,E1 24183.817,E2 24183.817} C_VEL
LIN {X 0,Y 512.487,Z 812.614,A -85,B 0,C 180,E1 24182.799,E2 24182.799} C_VEL
LIN {X 0,Y 513.456,Z 793.332,A -85,B 0,C 180,E1 24181.947,E2 24181.947} C_VEL
LIN {X 0,Y 514.273,Z 772.651,A -85,B 0,C 180,E1 24181.268,E2 24181.268} C_VEL
LIN {X 0,Y 514.803,Z 752.265,A -85,B 0,C 180,E1 24180.811,E2 24180.811} C_VEL
LIN {X 0,Y 517.544,Z 519.418,A -85,B 0,C 180,E1 24177.271,E2 24177.271} C_VEL
LIN {X 0,Y 511.919,Z 498.881,A -85,B 0,C 180,E1 24176.512,E2 24176.512} C_VEL
LIN {X 0,Y 512.543,Z 477.778,A -85,B 0,C 180,E1 24173.904,E2 24173.904} C_VEL
LIN {X 0,Y 507.296,Z 460.687,A -85,B 0,C 180,E1 24171.187,E2 24171.187} C_VEL
LIN {X 0,Y 504.674,Z 452.627,A -85,B 0,C 180,E1 24169.843,E2 24169.843} C_VEL
LIN {X 0,Y 504.692,Z 452.614,A -85,B 0,C 180,E1 24166.312,E2 24166.312} C_VEL
LIN {X 0,Y 504.705,Z 452.617,A -85,B 0,C 180,E1 24162.806,E2 24162.806} C_VEL
LIN {X 0,Y 504.71,Z 452.62,A -85,B 0,C 180,E1 24159.231,E2 24159.231} C_VEL
LIN {X 0,Y 504.697,Z 452.621,A -85,B 0,C 180,E1 24155.682,E2 24155.682} C_VEL
LIN {X 0,Y 504.706,Z 452.734,A -85,B 0,C 180,E1 24152.606,E2 24152.606} C_VEL
LIN {X 0,Y 512.499,Z 475.089,A -85,B 0,C 180,E1 24149.577,E2 24149.577} C_VEL
LIN {X 0,Y 513.819,Z 479.792,A -85,B 0,C 180,E1 24148.982,E2 24148.982} C_VEL
LIN {X 0,Y 512.503,Z 510.303,A -85,B 0,C 180,E1 24145.913,E2 24145.913} C_VEL
LIN {X 0,Y 511.118,Z 544.368,A -85,B 0,C 180,E1 24142.546,E2 24142.546} C_VEL
LIN {X 0,Y 509.71,Z 580.086,A -85,B 0,C 180,E1 24139.069,E2 24139.069} C_VEL
LIN {X 0,Y 508.813,Z 610.174,A -85,B 0,C 180,E1 24136.21,E2 24136.21} C_VEL
LIN {X 0,Y 509.447,Z 615.792,A -85,B 0,C 180,E1 24136.086,E2 24136.086} C_VEL
LIN {X 0,Y 507.763,Z 752.214,A -85,B 0,C 180,E1 24133.847,E2 24133.847} C_VEL
LIN {X 0,Y 507.546,Z 769.119,A -85,B 0,C 180,E1 24133.344,E2 24133.344} C_VEL
LIN {X 0,Y 507.229,Z 783.889,A -85,B 0,C 180,E1 24132.697,E2 24132.697} C_VEL
LIN {X 0,Y 506.795,Z 799.398,A -85,B 0,C 180,E1 24131.783,E2 24131.783} C_VEL
LIN {X 0,Y 506.34,Z 812.866,A -85,B 0,C 180,E1 24130.755,E2 24130.755} C_VEL
LIN {X 0,Y 505.839,Z 826.144,A -85,B 0,C 180,E1 24129.477,E2 24129.477} C_VEL
LIN {X 0,Y 505.393,Z 837.724,A -85,B 0,C 180,E1 24128.075,E2 24128.075} C_VEL
LIN {X 0,Y 505.005,Z 848.206,A -85,B 0,C 180,E1 24126.48,E2 24126.48} C_VEL
LIN {X 0,Y 504.724,Z 856.665,A -85,B 0,C 180,E1 24124.827,E2 24124.827} C_VEL
LIN {X 0,Y 504.526,Z 863.573,A -85,B 0,C 180,E1 24123.067,E2 24123.067} C_VEL
LIN {X 0,Y 504.4,Z 868.659,A -85,B 0,C 180,E1 24121.25,E2 24121.25} C_VEL
LIN {X 0,Y 504.356,Z 872.114,A -85,B 0,C 180,E1 24119.319,E2 24119.319} C_VEL
LIN {X 0,Y 504.337,Z 873.564,A -85,B 0,C 180,E1 24117.5,E2 24117.5} C_VEL
LIN {X 0,Y 504.378,Z 873.318,A -85,B 0,C 180,E1 24115.566,E2 24115.566} C_VEL
LIN {X 0,Y 504.433,Z 871.319,A -85,B 0,C 180,E1 24113.741,E2 24113.741} C_VEL
LIN {X 0,Y 504.575,Z 867.587,A -85,B 0,C 180,E1 24111.912,E2 24111.912} C_VEL
LIN {X 0,Y 504.77,Z 862.325,A -85,B 0,C 180,E1 24110.192,E2 24110.192} C_VEL
LIN {X 0,Y 505.048,Z 855.134,A -85,B 0,C 180,E1 24108.466,E2 24108.466} C_VEL
LIN {X 0,Y 505.392,Z 847.091,A -85,B 0,C 180,E1 24106.966,E2 24106.966} C_VEL
LIN {X 0,Y 505.824,Z 836.858,A -85,B 0,C 180,E1 24105.461,E2 24105.461} C_VEL
LIN {X 0,Y 506.298,Z 826.093,A -85,B 0,C 180,E1 24104.185,E2 24104.185} C_VEL
LIN {X 0,Y 506.77,Z 813.797,A -85,B 0,C 180,E1 24103.022,E2 24103.022} C_VEL
LIN {X 0,Y 507.226,Z 799.815,A -85,B 0,C 180,E1 24101.972,E2 24101.972} C_VEL
LIN {X 0,Y 507.565,Z 785.504,A -85,B 0,C 180,E1 24101.152,E2 24101.152} C_VEL
LIN {X 0,Y 507.814,Z 769.6,A -85,B 0,C 180,E1 24100.482,E2 24100.482} C_VEL
LIN {X 0,Y 507.888,Z 753.77,A -85,B 0,C 180,E1 24100.047,E2 24100.047} C_VEL
LIN {X 0,Y 509.602,Z 660.406,A -85,B 0,C 180,E1 24098.336,E2 24098.336} C_VEL
LIN {X 0,Y 510.777,Z 621.898,A -85,B 0,C 180,E1 24097.56,E2 24097.56} C_VEL
LIN {X 0,Y 512.538,Z 616.341,A -85,B 0,C 180,E1 24097.096,E2 24097.096} C_VEL
LIN {X 0,Y 515.813,Z 581.938,A -85,B 0,C 180,E1 24093.332,E2 24093.332} C_VEL
LIN {X 0,Y 520.088,Z 551.179,A -85,B 0,C 180,E1 24089.756,E2 24089.756} C_VEL
LIN {X 0,Y 525.116,Z 526.063,A -85,B 0,C 180,E1 24086.614,E2 24086.614} C_VEL
LIN {X 0,Y 529.016,Z 511.848,A -85,B 0,C 180,E1 24084.666,E2 24084.666} C_VEL
LIN {X 0,Y 531.426,Z 504.184,A -85,B 0,C 180,E1 24083.456,E2 24083.456} C_VEL
LIN {X 0,Y 531.001,Z 501.086,A -85,B 0,C 180,E1 24082.09,E2 24082.09} C_VEL
LIN {X 0,Y 531.165,Z 499.694,A -85,B 0,C 180,E1 24081.183,E2 24081.183} C_VEL
LIN {X 0,Y 531.589,Z 499.73,A -85,B 0,C 180,E1 24079.787,E2 24079.787} C_VEL
LIN {X 0,Y 531.696,Z 500.297,A -85,B 0,C 180,E1 24079.409,E2 24079.409} C_VEL
LIN {X 0,Y 525.988,Z 512.933,A -85,B 0,C 180,E1 24078.001,E2 24078.001} C_VEL
LIN {X 0,Y 521.372,Z 528.379,A -85,B 0,C 180,E1 24076.462,E2 24076.462} C_VEL
LIN {X 0,Y 517.622,Z 548.238,A -85,B 0,C 180,E1 24074.678,E2 24074.678} C_VEL
LIN {X 0,Y 516.329,Z 566.906,A -85,B 0,C 180,E1 24073.049,E2 24073.049} C_VEL
LIN {X 0,Y 517.174,Z 581.691,A -85,B 0,C 180,E1 24071.733,E2 24071.733} C_VEL
LIN {X 0,Y 519.963,Z 595.068,A -85,B 0,C 180,E1 24070.49,E2 24070.49} C_VEL
LIN {X 0,Y 524.381,Z 606.654,A -85,B 0,C 180,E1 24069.36,E2 24069.36} C_VEL
LIN {X 0,Y 530.292,Z 616.636,A -85,B 0,C 180,E1 24068.339,E2 24068.339} C_VEL
LIN {X 0,Y 538.192,Z 625.949,A -85,B 0,C 180,E1 24067.331,E2 24067.331} C_VEL
LIN {X 0,Y 547.041,Z 633.53,A -85,B 0,C 180,E1 24066.466,E2 24066.466} C_VEL
LIN {X 0,Y 557.388,Z 640.001,A -85,B 0,C 180,E1 24065.649,E2 24065.649} C_VEL
LIN {X 0,Y 566.513,Z 644.041,A -85,B 0,C 180,E1 24065.022,E2 24065.022} C_VEL
LIN {X 0,Y 571.644,Z 645.165,A -85,B 0,C 180,E1 24064.531,E2 24064.531} C_VEL
LIN {X 0,Y 575.349,Z 645.006,A -85,B 0,C 180,E1 24064.01,E2 24064.01} C_VEL
LIN {X 0,Y 576.359,Z 644.805,A -85,B 0,C 180,E1 24063.81,E2 24063.81} C_VEL
LIN {X 0,Y 567.08,Z 663.785,A -85,B 0,C 180,E1 24063.536,E2 24063.536} C_VEL
LIN {X 0,Y 556.913,Z 682.556,A -85,B 0,C 180,E1 24063.079,E2 24063.079} C_VEL
LIN {X 0,Y 550.196,Z 695.906,A -85,B 0,C 180,E1 24062.604,E2 24062.604} C_VEL
LIN {X 0,Y 537.489,Z 714.316,A -85,B 0,C 180,E1 24061.976,E2 24061.976} C_VEL
LIN {X 0,Y 529.509,Z 728.261,A -85,B 0,C 180,E1 24061.411,E2 24061.411} C_VEL
LIN {X 0,Y 524.035,Z 741.043,A -85,B 0,C 180,E1 24060.818,E2 24060.818} C_VEL
LIN {X 0,Y 521.359,Z 747.974,A -85,B 0,C 180,E1 24060.482,E2 24060.482} C_VEL
LIN {X 0,Y 517.233,Z 759.319,A -85,B 0,C 180,E1 24059.917,E2 24059.917} C_VEL
LIN {X 0,Y 514.362,Z 769.8,A -85,B 0,C 180,E1 24059.39,E2 24059.39} C_VEL
LIN {X 0,Y 513.759,Z 806.181,A -85,B 0,C 180,E1 24058.831,E2 24058.831} C_VEL
LIN {X 0,Y 513.122,Z 828.507,A -85,B 0,C 180,E1 24058.279,E2 24058.279} C_VEL
LIN {X 0,Y 512.383,Z 850.055,A -85,B 0,C 180,E1 24057.516,E2 24057.516} C_VEL
LIN {X 0,Y 511.546,Z 870.382,A -85,B 0,C 180,E1 24056.59,E2 24056.59} C_VEL
LIN {X 0,Y 510.59,Z 889.977,A -85,B 0,C 180,E1 24055.479,E2 24055.479} C_VEL
LIN {X 0,Y 509.759,Z 905.635,A -85,B 0,C 180,E1 24054.387,E2 24054.387} C_VEL
LIN {X 0,Y 508.686,Z 921.513,A -85,B 0,C 180,E1 24053.027,E2 24053.027} C_VEL
LIN {X 0,Y 507.495,Z 938.813,A -85,B 0,C 180,E1 24051.255,E2 24051.255} C_VEL
LIN {X 0,Y 506.65,Z 951.555,A -85,B 0,C 180,E1 24049.722,E2 24049.722} C_VEL
LIN {X 0,Y 505.827,Z 965.095,A -85,B 0,C 180,E1 24047.842,E2 24047.842} C_VEL
LIN {X 0,Y 505.142,Z 977.061,A -85,B 0,C 180,E1 24045.853,E2 24045.853} C_VEL
LIN {X 0,Y 504.642,Z 987.799,A -85,B 0,C 180,E1 24043.755,E2 24043.755} C_VEL
LIN {X 0,Y 504.282,Z 996.939,A -85,B 0,C 180,E1 24041.553,E2 24041.553} C_VEL
LIN {X 0,Y 504.073,Z 1004.36,A -85,B 0,C 180,E1 24039.361,E2 24039.361} C_VEL
LIN {X 0,Y 503.96,Z 1009.971,A -85,B 0,C 180,E1 24037.181,E2 24037.181} C_VEL
LIN {X 0,Y 503.918,Z 1013.973,A -85,B 0,C 180,E1 24035.095,E2 24035.095} C_VEL
LIN {X 0,Y 503.911,Z 1016.818,A -85,B 0,C 180,E1 24032.73,E2 24032.73} C_VEL
LIN {X 0,Y 503.901,Z 1017.887,A -85,B 0,C 180,E1 24030.569,E2 24030.569} C_VEL
LIN {X 0,Y 503.909,Z 1017.47,A -85,B 0,C 180,E1 24028.181,E2 24028.181} C_VEL
LIN {X 0,Y 503.92,Z 1015.369,A -85,B 0,C 180,E1 24025.904,E2 24025.904} C_VEL
LIN {X 0,Y 503.953,Z 1011.737,A -85,B 0,C 180,E1 24023.622,E2 24023.622} C_VEL
LIN {X 0,Y 504.034,Z 1006.581,A -85,B 0,C 180,E1 24021.444,E2 24021.444} C_VEL
LIN {X 0,Y 504.197,Z 999.925,A -85,B 0,C 180,E1 24019.257,E2 24019.257} C_VEL
LIN {X 0,Y 504.49,Z 991.354,A -85,B 0,C 180,E1 24017.059,E2 24017.059} C_VEL
LIN {X 0,Y 504.891,Z 982.084,A -85,B 0,C 180,E1 24015.082,E2 24015.082} C_VEL
LIN {X 0,Y 505.515,Z 970.25,A -85,B 0,C 180,E1 24012.979,E2 24012.979} C_VEL
LIN {X 0,Y 506.208,Z 958.587,A -85,B 0,C 180,E1 24011.219,E2 24011.219} C_VEL
LIN {X 0,Y 507.193,Z 943.443,A -85,B 0,C 180,E1 24009.278,E2 24009.278} C_VEL
LIN {X 0,Y 508.137,Z 929.369,A -85,B 0,C 180,E1 24007.742,E2 24007.742} C_VEL
LIN {X 0,Y 509.302,Z 912.68,A -85,B 0,C 180,E1 24006.184,E2 24006.184} C_VEL
LIN {X 0,Y 510.275,Z 896.735,A -85,B 0,C 180,E1 24004.961,E2 24004.961} C_VEL
LIN {X 0,Y 511.315,Z 877.214,A -85,B 0,C 180,E1 24003.734,E2 24003.734} C_VEL
LIN {X 0,Y 512.322,Z 856.989,A -85,B 0,C 180,E1 24002.702,E2 24002.702} C_VEL
LIN {X 0,Y 513.205,Z 835.818,A -85,B 0,C 180,E1 24001.858,E2 24001.858} C_VEL
LIN {X 0,Y 513.95,Z 814.34,A -85,B 0,C 180,E1 24001.229,E2 24001.229} C_VEL
LIN {X 0,Y 514.455,Z 792.205,A -85,B 0,C 180,E1 24000.805,E2 24000.805} C_VEL
LIN {X 0,Y 514.822,Z 770.306,A -85,B 0,C 180,E1 24000.475,E2 24000.475} C_VEL
LIN {X 0,Y 520.172,Z 752.744,A -85,B 0,C 180,E1 23999.57,E2 23999.57} C_VEL
LIN {X 0,Y 524.05,Z 743.025,A -85,B 0,C 180,E1 23999.121,E2 23999.121} C_VEL
LIN {X 0,Y 529.038,Z 730.657,A -85,B 0,C 180,E1 23998.559,E2 23998.559} C_VEL
LIN {X 0,Y 536.899,Z 716.048,A -85,B 0,C 180,E1 23998.007,E2 23998.007} C_VEL
LIN {X 0,Y 549.599,Z 696.755,A -85,B 0,C 180,E1 23997.419,E2 23997.419} C_VEL
LIN {X 0,Y 551.55,Z 693.325,A -85,B 0,C 180,E1 23997.302,E2 23997.302} C_VEL
LIN {X 0,Y 557.902,Z 680.722,A -85,B 0,C 180,E1 23996.866,E2 23996.866} C_VEL
LIN {X 0,Y 568.168,Z 661.702,A -85,B 0,C 180,E1 23996.426,E2 23996.426} C_VEL
LIN {X 0,Y 576.348,Z 644.718,A -85,B 0,C 180,E1 23996.177,E2 23996.177} C_VEL
LIN {X 0,Y 572.953,Z 645.243,A -85,B 0,C 180,E1 23995.632,E2 23995.632} C_VEL
LIN {X 0,Y 568.183,Z 644.53,A -85,B 0,C 180,E1 23995.117,E2 23995.117} C_VEL
LIN {X 0,Y 557.258,Z 640.299,A -85,B 0,C 180,E1 23994.193,E2 23994.193} C_VEL
LIN {X 0,Y 547.949,Z 634.793,A -85,B 0,C 180,E1 23993.231,E2 23993.231} C_VEL
LIN {X 0,Y 539.556,Z 627.622,A -85,B 0,C 180,E1 23992.166,E2 23992.166} C_VEL
LIN {X 0,Y 532.992,Z 619.587,A -85,B 0,C 180,E1 23991.124,E2 23991.124} C_VEL
LIN {X 0,Y 527.456,Z 609.666,A -85,B 0,C 180,E1 23989.981,E2 23989.981} C_VEL
LIN {X 0,Y 523.41,Z 597.885,A -85,B 0,C 180,E1 23988.774,E2 23988.774} C_VEL
LIN {X 0,Y 520.86,Z 583.958,A -85,B 0,C 180,E1 23987.488,E2 23987.488} C_VEL
LIN {X 0,Y 520.048,Z 566.671,A -85,B 0,C 180,E1 23986.048,E2 23986.048} C_VEL
LIN {X 0,Y 522.987,Z 514.121,A -85,B 0,C 180,E1 23982,E2 23982} C_VEL
LIN {X 0,Y 524.301,Z 493.181,A -85,B 0,C 180,E1 23980.348,E2 23980.348} C_VEL
LIN {X 0,Y 514.903,Z 473.658,A -85,B 0,C 180,E1 23977.57,E2 23977.57} C_VEL
LIN {X 0,Y 508.407,Z 460.799,A -85,B 0,C 180,E1 23975.6,E2 23975.6} C_VEL
LIN {X 0,Y 506.313,Z 456.551,A -85,B 0,C 180,E1 23974.938,E2 23974.938} C_VEL
LIN {X 0,Y 504.804,Z 453.183,A -85,B 0,C 180,E1 23974.419,E2 23974.419} C_VEL
LIN {X 0,Y 504.712,Z 452.609,A -85,B 0,C 180,E1 23974.301,E2 23974.301} C_VEL
LIN {X 0,Y 504.681,Z 452.621,A -85,B 0,C 180,E1 23970.74,E2 23970.74} C_VEL
LIN {X 0,Y 504.662,Z 452.622,A -85,B 0,C 180,E1 23967.109,E2 23967.109} C_VEL
LIN {X 0,Y 504.708,Z 452.617,A -85,B 0,C 180,E1 23963.589,E2 23963.589} C_VEL
LIN {X 0,Y 504.666,Z 452.623,A -85,B 0,C 180,E1 23960.165,E2 23960.165} C_VEL
LIN {X 0,Y 504.694,Z 452.621,A -85,B 0,C 180,E1 23956.694,E2 23956.694} C_VEL
LIN {X 0,Y 504.709,Z 452.619,A -85,B 0,C 180,E1 23953.169,E2 23953.169} C_VEL
LIN {X 0,Y 504.711,Z 452.618,A -85,B 0,C 180,E1 23949.464,E2 23949.464} C_VEL
LIN {X 0,Y 504.684,Z 452.62,A -85,B 0,C 180,E1 23945.913,E2 23945.913} C_VEL
LIN {X 0,Y 504.656,Z 452.622,A -85,B 0,C 180,E1 23942.384,E2 23942.384} C_VEL
LIN {X 0,Y 504.709,Z 452.615,A -85,B 0,C 180,E1 23938.978,E2 23938.978} C_VEL
LIN {X 0,Y 504.656,Z 452.62,A -85,B 0,C 180,E1 23935.568,E2 23935.568} C_VEL
LIN {X 0,Y 504.681,Z 452.609,A -85,B 0,C 180,E1 23932.028,E2 23932.028} C_VEL
LIN {X 0,Y 504.709,Z 452.616,A -85,B 0,C 180,E1 23928.574,E2 23928.574} C_VEL
LIN {X 0,Y 504.695,Z 452.619,A -85,B 0,C 180,E1 23924.958,E2 23924.958} C_VEL
LIN {X 0,Y 504.704,Z 452.611,A -85,B 0,C 180,E1 23921.52,E2 23921.52} C_VEL
LIN {X 0,Y 504.683,Z 452.613,A -85,B 0,C 180,E1 23917.998,E2 23917.998} C_VEL
LIN {X 0,Y 504.706,Z 452.616,A -85,B 0,C 180,E1 23914.539,E2 23914.539} C_VEL
LIN {X 0,Y 504.669,Z 452.623,A -85,B 0,C 180,E1 23911.091,E2 23911.091} C_VEL
LIN {X 0,Y 504.685,Z 452.62,A -85,B 0,C 180,E1 23907.527,E2 23907.527} C_VEL
LIN {X 0,Y 504.694,Z 452.618,A -85,B 0,C 180,E1 23904.097,E2 23904.097} C_VEL
LIN {X 0,Y 504.658,Z 452.623,A -85,B 0,C 180,E1 23900.595,E2 23900.595} C_VEL
LIN {X 0,Y 504.7,Z 452.62,A -85,B 0,C 180,E1 23897.039,E2 23897.039} C_VEL
LIN {X 0,Y 504.694,Z 452.619,A -85,B 0,C 180,E1 23893.584,E2 23893.584} C_VEL
LIN {X 0,Y 504.704,Z 452.617,A -85,B 0,C 180,E1 23890.088,E2 23890.088} C_VEL
LIN {X 0,Y 503.826,Z 453.017,A -85,B 0,C 180,E1 23889.479,E2 23889.479} C_VEL
LIN {X 0,Y 501.049,Z 454.87,A -85,B 0,C 180,E1 23888.664,E2 23888.664} C_VEL
LIN {X 0,Y 499.321,Z 457.454,A -85,B 0,C 180,E1 23888.057,E2 23888.057} C_VEL
LIN {X 0,Y 499.27,Z 460.075,A -85,B 0,C 180,E1 23887.637,E2 23887.637} C_VEL
LIN {X 0,Y 499.428,Z 460.561,A -85,B 0,C 180,E1 23887.574,E2 23887.574} C_VEL
LIN {X 0,Y 507.544,Z 482.196,A -85,B 0,C 180,E1 23884.963,E2 23884.963} C_VEL
LIN {X 0,Y 507.947,Z 484.415,A -85,B 0,C 180,E1 23884.74,E2 23884.74} C_VEL
LIN {X 0,Y 507.673,Z 497.368,A -85,B 0,C 180,E1 23883.731,E2 23883.731} C_VEL
LIN {X 0,Y 510.988,Z 515.722,A -85,B 0,C 180,E1 23883.177,E2 23883.177} C_VEL
LIN {X 0,Y 507.739,Z 756.84,A -85,B 0,C 180,E1 23879.455,E2 23879.455} C_VEL
LIN {X 0,Y 507.05,Z 777.792,A -85,B 0,C 180,E1 23878.933,E2 23878.933} C_VEL
LIN {X 0,Y 506.169,Z 797.99,A -85,B 0,C 180,E1 23878.209,E2 23878.209} C_VEL
LIN {X 0,Y 505.131,Z 816.694,A -85,B 0,C 180,E1 23877.336,E2 23877.336} C_VEL
LIN {X 0,Y 503.961,Z 835.142,A -85,B 0,C 180,E1 23876.258,E2 23876.258} C_VEL
LIN {X 0,Y 502.645,Z 853.477,A -85,B 0,C 180,E1 23874.942,E2 23874.942} C_VEL
LIN {X 0,Y 501.363,Z 870.098,A -85,B 0,C 180,E1 23873.506,E2 23873.506} C_VEL
LIN {X 0,Y 500.141,Z 885.818,A -85,B 0,C 180,E1 23871.897,E2 23871.897} C_VEL
LIN {X 0,Y 498.945,Z 901.748,A -85,B 0,C 180,E1 23869.973,E2 23869.973} C_VEL
LIN {X 0,Y 498.004,Z 915.529,A -85,B 0,C 180,E1 23868.01,E2 23868.01} C_VEL
LIN {X 0,Y 497.267,Z 927.521,A -85,B 0,C 180,E1 23865.989,E2 23865.989} C_VEL
LIN {X 0,Y 496.71,Z 938.128,A -85,B 0,C 180,E1 23863.859,E2 23863.859} C_VEL
LIN {X 0,Y 496.326,Z 947.277,A -85,B 0,C 180,E1 23861.621,E2 23861.621} C_VEL
LIN {X 0,Y 496.088,Z 954.54,A -85,B 0,C 180,E1 23859.395,E2 23859.395} C_VEL
LIN {X 0,Y 495.963,Z 960.4,A -85,B 0,C 180,E1 23857.063,E2 23857.063} C_VEL
LIN {X 0,Y 495.924,Z 964.547,A -85,B 0,C 180,E1 23854.741,E2 23854.741} C_VEL
LIN {X 0,Y 495.91,Z 967.076,A -85,B 0,C 180,E1 23852.426,E2 23852.426} C_VEL
LIN {X 0,Y 495.913,Z 967.976,A -85,B 0,C 180,E1 23850.115,E2 23850.115} C_VEL
LIN {X 0,Y 495.911,Z 967.263,A -85,B 0,C 180,E1 23847.804,E2 23847.804} C_VEL
LIN {X 0,Y 495.922,Z 964.828,A -85,B 0,C 180,E1 23845.374,E2 23845.374} C_VEL
LIN {X 0,Y 495.965,Z 960.591,A -85,B 0,C 180,E1 23842.936,E2 23842.936} C_VEL
LIN {X 0,Y 496.071,Z 955.151,A -85,B 0,C 180,E1 23840.72,E2 23840.72} C_VEL
LIN {X 0,Y 496.312,Z 947.604,A -85,B 0,C 180,E1 23838.377,E2 23838.377} C_VEL
LIN {X 0,Y 496.693,Z 938.514,A -85,B 0,C 180,E1 23836.139,E2 23836.139} C_VEL
LIN {X 0,Y 497.248,Z 927.827,A -85,B 0,C 180,E1 23833.979,E2 23833.979} C_VEL
LIN {X 0,Y 497.965,Z 916.086,A -85,B 0,C 180,E1 23831.987,E2 23831.987} C_VEL
LIN {X 0,Y 498.933,Z 901.916,A -85,B 0,C 180,E1 23829.959,E2 23829.959} C_VEL
LIN {X 0,Y 500.162,Z 885.57,A -85,B 0,C 180,E1 23827.986,E2 23827.986} C_VEL
LIN {X 0,Y 501.445,Z 869.075,A -85,B 0,C 180,E1 23826.31,E2 23826.31} C_VEL
LIN {X 0,Y 502.726,Z 852.226,A -85,B 0,C 180,E1 23824.872,E2 23824.872} C_VEL
LIN {X 0,Y 503.997,Z 834.57,A -85,B 0,C 180,E1 23823.615,E2 23823.615} C_VEL
LIN {X 0,Y 505.176,Z 816.034,A -85,B 0,C 180,E1 23822.537,E2 23822.537} C_VEL
LIN {X 0,Y 506.208,Z 797.255,A -85,B 0,C 180,E1 23821.67,E2 23821.67} C_VEL
LIN {X 0,Y 507.08,Z 777.032,A -85,B 0,C 180,E1 23820.955,E2 23820.955} C_VEL
LIN {X 0,Y 507.756,Z 756.027,A -85,B 0,C 180,E1 23820.439,E2 23820.439} C_VEL
LIN {X 0,Y 510.822,Z 521.182,A -85,B 0,C 180,E1 23816.811,E2 23816.811} C_VEL
LIN {X 0,Y 504.759,Z 498.998,A -85,B 0,C 180,E1 23815.971,E2 23815.971} C_VEL
LIN {X 0,Y 505.329,Z 480.959,A -85,B 0,C 180,E1 23813.728,E2 23813.728} C_VEL
LIN {X 0,Y 500.216,Z 464.231,A -85,B 0,C 180,E1 23811.037,E2 23811.037} C_VEL
LIN {X 0,Y 496.768,Z 453.612,A -85,B 0,C 180,E1 23809.254,E2 23809.254} C_VEL
LIN {X 0,Y 496.742,Z 453.606,A -85,B 0,C 180,E1 23805.696,E2 23805.696} C_VEL
LIN {X 0,Y 496.754,Z 453.604,A -85,B 0,C 180,E1 23802.087,E2 23802.087} C_VEL
LIN {X 0,Y 496.762,Z 453.607,A -85,B 0,C 180,E1 23798.606,E2 23798.606} C_VEL
LIN {X 0,Y 496.761,Z 453.613,A -85,B 0,C 180,E1 23794.995,E2 23794.995} C_VEL
LIN {X 0,Y 496.776,Z 453.678,A -85,B 0,C 180,E1 23793.193,E2 23793.193} C_VEL
LIN {X 0,Y 504.992,Z 477.084,A -85,B 0,C 180,E1 23789.964,E2 23789.964} C_VEL
LIN {X 0,Y 506.671,Z 482.24,A -85,B 0,C 180,E1 23789.279,E2 23789.279} C_VEL
LIN {X 0,Y 505.277,Z 512.787,A -85,B 0,C 180,E1 23786.186,E2 23786.186} C_VEL
LIN {X 0,Y 503.771,Z 547.028,A -85,B 0,C 180,E1 23782.77,E2 23782.77} C_VEL
LIN {X 0,Y 502.291,Z 582.402,A -85,B 0,C 180,E1 23779.296,E2 23779.296} C_VEL
LIN {X 0,Y 501.352,Z 611.074,A -85,B 0,C 180,E1 23776.542,E2 23776.542} C_VEL
LIN {X 0,Y 502.013,Z 616.722,A -85,B 0,C 180,E1 23776.41,E2 23776.41} C_VEL
LIN {X 0,Y 500.134,Z 753.366,A -85,B 0,C 180,E1 23774.102,E2 23774.102} C_VEL
LIN {X 0,Y 499.908,Z 770.143,A -85,B 0,C 180,E1 23773.593,E2 23773.593} C_VEL
LIN {X 0,Y 499.553,Z 785.501,A -85,B 0,C 180,E1 23772.904,E2 23772.904} C_VEL
LIN {X 0,Y 499.093,Z 801.016,A -85,B 0,C 180,E1 23771.967,E2 23771.967} C_VEL
LIN {X 0,Y 498.603,Z 814.352,A -85,B 0,C 180,E1 23770.924,E2 23770.924} C_VEL
LIN {X 0,Y 498.076,Z 827.354,A -85,B 0,C 180,E1 23769.65,E2 23769.65} C_VEL
LIN {X 0,Y 497.624,Z 838.264,A -85,B 0,C 180,E1 23768.318,E2 23768.318} C_VEL
LIN {X 0,Y 497.195,Z 848.865,A -85,B 0,C 180,E1 23766.698,E2 23766.698} C_VEL
LIN {X 0,Y 496.887,Z 857.211,A -85,B 0,C 180,E1 23765.08,E2 23765.08} C_VEL
LIN {X 0,Y 496.654,Z 864.483,A -85,B 0,C 180,E1 23763.232,E2 23763.232} C_VEL
LIN {X 0,Y 496.517,Z 869.443,A -85,B 0,C 180,E1 23761.5,E2 23761.5} C_VEL
LIN {X 0,Y 496.456,Z 873.074,A -85,B 0,C 180,E1 23759.539,E2 23759.539} C_VEL
LIN {X 0,Y 496.439,Z 874.77,A -85,B 0,C 180,E1 23757.692,E2 23757.692} C_VEL
LIN {X 0,Y 496.476,Z 874.689,A -85,B 0,C 180,E1 23755.727,E2 23755.727} C_VEL
LIN {X 0,Y 496.548,Z 872.921,A -85,B 0,C 180,E1 23753.874,E2 23753.874} C_VEL
LIN {X 0,Y 496.707,Z 869.081,A -85,B 0,C 180,E1 23751.9,E2 23751.9} C_VEL
LIN {X 0,Y 496.93,Z 863.924,A -85,B 0,C 180,E1 23750.153,E2 23750.153} C_VEL
LIN {X 0,Y 497.261,Z 856.386,A -85,B 0,C 180,E1 23748.304,E2 23748.304} C_VEL
LIN {X 0,Y 497.645,Z 848.18,A -85,B 0,C 180,E1 23746.759,E2 23746.759} C_VEL
LIN {X 0,Y 498.129,Z 837.907,A -85,B 0,C 180,E1 23745.231,E2 23745.231} C_VEL
LIN {X 0,Y 498.643,Z 827.045,A -85,B 0,C 180,E1 23743.936,E2 23743.936} C_VEL
LIN {X 0,Y 499.178,Z 813.962,A -85,B 0,C 180,E1 23742.696,E2 23742.696} C_VEL
LIN {X 0,Y 499.648,Z 800.56,A -85,B 0,C 180,E1 23741.689,E2 23741.689} C_VEL
LIN {X 0,Y 500.012,Z 786.067,A -85,B 0,C 180,E1 23740.856,E2 23740.856} C_VEL
LIN {X 0,Y 500.265,Z 770.721,A -85,B 0,C 180,E1 23740.205,E2 23740.205} C_VEL
LIN {X 0,Y 500.326,Z 754.421,A -85,B 0,C 180,E1 23739.759,E2 23739.759} C_VEL
LIN {X 0,Y 502.054,Z 671.234,A -85,B 0,C 180,E1 23738.162,E2 23738.162} C_VEL
LIN {X 0,Y 503.613,Z 624.709,A -85,B 0,C 180,E1 23737.192,E2 23737.192} C_VEL
LIN {X 0,Y 505.791,Z 618.23,A -85,B 0,C 180,E1 23736.65,E2 23736.65} C_VEL
LIN {X 0,Y 509.343,Z 584.737,A -85,B 0,C 180,E1 23732.908,E2 23732.908} C_VEL
LIN {X 0,Y 514.065,Z 554.29,A -85,B 0,C 180,E1 23729.283,E2 23729.283} C_VEL
LIN {X 0,Y 519.447,Z 530.322,A -85,B 0,C 180,E1 23726.201,E2 23726.201} C_VEL
LIN {X 0,Y 523.966,Z 515.805,A -85,B 0,C 180,E1 23724.138,E2 23724.138} C_VEL
LIN {X 0,Y 526.148,Z 509.633,A -85,B 0,C 180,E1 23723.094,E2 23723.094} C_VEL
LIN {X 0,Y 526.071,Z 507.088,A -85,B 0,C 180,E1 23721.852,E2 23721.852} C_VEL
LIN {X 0,Y 526.342,Z 505.999,A -85,B 0,C 180,E1 23720.983,E2 23720.983} C_VEL
LIN {X 0,Y 526.802,Z 506.142,A -85,B 0,C 180,E1 23719.811,E2 23719.811} C_VEL
LIN {X 0,Y 520.488,Z 518.777,A -85,B 0,C 180,E1 23718.355,E2 23718.355} C_VEL
LIN {X 0,Y 515.51,Z 533.556,A -85,B 0,C 180,E1 23716.826,E2 23716.826} C_VEL
LIN {X 0,Y 511.417,Z 552.442,A -85,B 0,C 180,E1 23715.052,E2 23715.052} C_VEL
LIN {X 0,Y 509.854,Z 570.26,A -85,B 0,C 180,E1 23713.422,E2 23713.422} C_VEL
LIN {X 0,Y 510.465,Z 584.922,A -85,B 0,C 180,E1 23712.059,E2 23712.059} C_VEL
LIN {X 0,Y 513.18,Z 598.769,A -85,B 0,C 180,E1 23710.72,E2 23710.72} C_VEL
LIN {X 0,Y 517.681,Z 610.831,A -85,B 0,C 180,E1 23709.502,E2 23709.502} C_VEL
LIN {X 0,Y 523.448,Z 620.779,A -85,B 0,C 180,E1 23708.45,E2 23708.45} C_VEL
LIN {X 0,Y 531.19,Z 630.207,A -85,B 0,C 180,E1 23707.408,E2 23707.408} C_VEL
LIN {X 0,Y 539.877,Z 638.001,A -85,B 0,C 180,E1 23706.508,E2 23706.508} C_VEL
LIN {X 0,Y 550.9,Z 645.275,A -85,B 0,C 180,E1 23705.6,E2 23705.6} C_VEL
LIN {X 0,Y 562.609,Z 650.701,A -85,B 0,C 180,E1 23704.809,E2 23704.809} C_VEL
LIN {X 0,Y 567.869,Z 652.257,A -85,B 0,C 180,E1 23704.361,E2 23704.361} C_VEL
LIN {X 0,Y 556.75,Z 670.277,A -85,B 0,C 180,E1 23703.886,E2 23703.886} C_VEL
LIN {X 0,Y 546.843,Z 687.08,A -85,B 0,C 180,E1 23703.267,E2 23703.267} C_VEL
LIN {X 0,Y 543.403,Z 693.653,A -85,B 0,C 180,E1 23703.001,E2 23703.001} C_VEL
LIN {X 0,Y 530.624,Z 712.092,A -85,B 0,C 180,E1 23702.354,E2 23702.354} C_VEL
LIN {X 0,Y 522.361,Z 726.59,A -85,B 0,C 180,E1 23701.762,E2 23701.762} C_VEL
LIN {X 0,Y 516.855,Z 739.372,A -85,B 0,C 180,E1 23701.164,E2 23701.164} C_VEL
LIN {X 0,Y 514.172,Z 746.31,A -85,B 0,C 180,E1 23700.825,E2 23700.825} C_VEL
LIN {X 0,Y 509.713,Z 758.55,A -85,B 0,C 180,E1 23700.21,E2 23700.21} C_VEL
LIN {X 0,Y 507.628,Z 765.891,A -85,B 0,C 180,E1 23699.853,E2 23699.853} C_VEL
LIN {X 0,Y 507.017,Z 779.237,A -85,B 0,C 180,E1 23699.68,E2 23699.68} C_VEL
LIN {X 0,Y 506.518,Z 808.88,A -85,B 0,C 180,E1 23699.178,E2 23699.178} C_VEL
LIN {X 0,Y 505.801,Z 829.234,A -85,B 0,C 180,E1 23698.632,E2 23698.632} C_VEL
LIN {X 0,Y 504.957,Z 848.92,A -85,B 0,C 180,E1 23697.892,E2 23697.892} C_VEL
LIN {X 0,Y 503.94,Z 868.075,A -85,B 0,C 180,E1 23696.96,E2 23696.96} C_VEL
LIN {X 0,Y 502.636,Z 892.451,A -85,B 0,C 180,E1 23695.511,E2 23695.511} C_VEL
LIN {X 0,Y 501.612,Z 910.896,A -85,B 0,C 180,E1 23694.182,E2 23694.182} C_VEL
LIN {X 0,Y 500.564,Z 928.256,A -85,B 0,C 180,E1 23692.676,E2 23692.676} C_VEL
LIN {X 0,Y 499.755,Z 940.329,A -85,B 0,C 180,E1 23691.416,E2 23691.416} C_VEL
LIN {X 0,Y 498.887,Z 952.457,A -85,B 0,C 180,E1 23689.921,E2 23689.921} C_VEL
LIN {X 0,Y 497.989,Z 965.841,A -85,B 0,C 180,E1 23688.012,E2 23688.012} C_VEL
LIN {X 0,Y 497.284,Z 977.057,A -85,B 0,C 180,E1 23686.11,E2 23686.11} C_VEL
LIN {X 0,Y 496.735,Z 987.597,A -85,B 0,C 180,E1 23684.024,E2 23684.024} C_VEL
LIN {X 0,Y 496.345,Z 996.498,A -85,B 0,C 180,E1 23681.858,E2 23681.858} C_VEL
LIN {X 0,Y 496.116,Z 1003.645,A -85,B 0,C 180,E1 23679.747,E2 23679.747} C_VEL
LIN {X 0,Y 495.972,Z 1009.718,A -85,B 0,C 180,E1 23677.414,E2 23677.414} C_VEL
LIN {X 0,Y 495.919,Z 1013.727,A -85,B 0,C 180,E1 23675.322,E2 23675.322} C_VEL
LIN {X 0,Y 495.91,Z 1016.731,A -85,B 0,C 180,E1 23672.89,E2 23672.89} C_VEL
LIN {X 0,Y 495.904,Z 1017.856,A -85,B 0,C 180,E1 23670.694,E2 23670.694} C_VEL
LIN {X 0,Y 495.902,Z 1017.605,A -85,B 0,C 180,E1 23668.383,E2 23668.383} C_VEL
LIN {X 0,Y 495.918,Z 1015.641,A -85,B 0,C 180,E1 23666.07,E2 23666.07} C_VEL
LIN {X 0,Y 495.95,Z 1012.367,A -85,B 0,C 180,E1 23663.867,E2 23663.867} C_VEL
LIN {X 0,Y 496.036,Z 1007.202,A -85,B 0,C 180,E1 23661.539,E2 23661.539} C_VEL
LIN {X 0,Y 496.191,Z 1001.044,A -85,B 0,C 180,E1 23659.434,E2 23659.434} C_VEL
LIN {X 0,Y 496.522,Z 992.291,A -85,B 0,C 180,E1 23657.069,E2 23657.069} C_VEL
LIN {X 0,Y 496.942,Z 983.234,A -85,B 0,C 180,E1 23655.077,E2 23655.077} C_VEL
LIN {X 0,Y 497.614,Z 971.711,A -85,B 0,C 180,E1 23652.941,E2 23652.941} C_VEL
LIN {X 0,Y 498.346,Z 960.225,A -85,B 0,C 180,E1 23651.155,E2 23651.155} C_VEL
LIN {X 0,Y 499.339,Z 946.49,A -85,B 0,C 180,E1 23649.304,E2 23649.304} C_VEL
LIN {X 0,Y 500.253,Z 933.131,A -85,B 0,C 180,E1 23647.806,E2 23647.806} C_VEL
LIN {X 0,Y 501.327,Z 916.81,A -85,B 0,C 180,E1 23646.268,E2 23646.268} C_VEL
LIN {X 0,Y 502.49,Z 898.179,A -85,B 0,C 180,E1 23644.798,E2 23644.798} C_VEL
LIN {X 0,Y 503.628,Z 878.886,A -85,B 0,C 180,E1 23643.532,E2 23643.532} C_VEL
LIN {X 0,Y 504.684,Z 859.857,A -85,B 0,C 180,E1 23642.51,E2 23642.51} C_VEL
LIN {X 0,Y 505.659,Z 839.372,A -85,B 0,C 180,E1 23641.632,E2 23641.632} C_VEL
LIN {X 0,Y 506.508,Z 818.587,A -85,B 0,C 180,E1 23640.97,E2 23640.97} C_VEL
LIN {X 0,Y 507.126,Z 797.496,A -85,B 0,C 180,E1 23640.508,E2 23640.508} C_VEL
LIN {X 0,Y 507.755,Z 769.16,A -85,B 0,C 180,E1 23640.055,E2 23640.055} C_VEL
LIN {X 0,Y 513.064,Z 752.058,A -85,B 0,C 180,E1 23639.168,E2 23639.168} C_VEL
LIN {X 0,Y 517.281,Z 741.445,A -85,B 0,C 180,E1 23638.672,E2 23638.672} C_VEL
LIN {X 0,Y 522.777,Z 728.218,A -85,B 0,C 180,E1 23638.074,E2 23638.074} C_VEL
LIN {X 0,Y 531.066,Z 713.066,A -85,B 0,C 180,E1 23637.508,E2 23637.508} C_VEL
LIN {X 0,Y 544.961,Z 691.768,A -85,B 0,C 180,E1 23636.856,E2 23636.856} C_VEL
LIN {X 0,Y 552.199,Z 677.947,A -85,B 0,C 180,E1 23636.354,E2 23636.354} C_VEL
LIN {X 0,Y 565.416,Z 656.338,A -85,B 0,C 180,E1 23635.728,E2 23635.728} C_VEL
LIN {X 0,Y 567.944,Z 652.129,A -85,B 0,C 180,E1 23635.636,E2 23635.636} C_VEL
LIN {X 0,Y 561.838,Z 650.46,A -85,B 0,C 180,E1 23635.125,E2 23635.125} C_VEL
LIN {X 0,Y 551.105,Z 645.918,A -85,B 0,C 180,E1 23634.192,E2 23634.192} C_VEL
LIN {X 0,Y 541.184,Z 639.686,A -85,B 0,C 180,E1 23633.128,E2 23633.128} C_VEL
LIN {X 0,Y 532.658,Z 631.962,A -85,B 0,C 180,E1 23631.998,E2 23631.998} C_VEL
LIN {X 0,Y 525.889,Z 623.207,A -85,B 0,C 180,E1 23630.87,E2 23630.87} C_VEL
LIN {X 0,Y 520.503,Z 613.011,A -85,B 0,C 180,E1 23629.695,E2 23629.695} C_VEL
LIN {X 0,Y 516.496,Z 600.685,A -85,B 0,C 180,E1 23628.427,E2 23628.427} C_VEL
LIN {X 0,Y 514.063,Z 586.419,A -85,B 0,C 180,E1 23627.098,E2 23627.098} C_VEL
LIN {X 0,Y 513.372,Z 568.914,A -85,B 0,C 180,E1 23625.625,E2 23625.625} C_VEL
LIN {X 0,Y 516.513,Z 516.839,A -85,B 0,C 180,E1 23621.576,E2 23621.576} C_VEL
LIN {X 0,Y 517.87,Z 497.215,A -85,B 0,C 180,E1 23620.01,E2 23620.01} C_VEL
LIN {X 0,Y 508.649,Z 478.119,A -85,B 0,C 180,E1 23617.26,E2 23617.26} C_VEL
LIN {X 0,Y 500.468,Z 461.736,A -85,B 0,C 180,E1 23614.707,E2 23614.707} C_VEL
LIN {X 0,Y 498.405,Z 457.545,A -85,B 0,C 180,E1 23614.035,E2 23614.035} C_VEL
LIN {X 0,Y 496.89,Z 454.401,A -85,B 0,C 180,E1 23613.529,E2 23613.529} C_VEL
LIN {X 0,Y 496.752,Z 453.609,A -85,B 0,C 180,E1 23613.394,E2 23613.394} C_VEL
LIN {X 0,Y 496.775,Z 453.606,A -85,B 0,C 180,E1 23609.811,E2 23609.811} C_VEL
LIN {X 0,Y 496.773,Z 453.606,A -85,B 0,C 180,E1 23606.148,E2 23606.148} C_VEL
LIN {X 0,Y 496.746,Z 453.61,A -85,B 0,C 180,E1 23602.609,E2 23602.609} C_VEL
LIN {X 0,Y 496.723,Z 453.612,A -85,B 0,C 180,E1 23599.032,E2 23599.032} C_VEL
LIN {X 0,Y 496.769,Z 453.606,A -85,B 0,C 180,E1 23595.647,E2 23595.647} C_VEL
LIN {X 0,Y 496.717,Z 453.612,A -85,B 0,C 180,E1 23592.202,E2 23592.202} C_VEL
LIN {X 0,Y 496.747,Z 453.608,A -85,B 0,C 180,E1 23588.566,E2 23588.566} C_VEL
LIN {X 0,Y 496.771,Z 453.607,A -85,B 0,C 180,E1 23585.081,E2 23585.081} C_VEL
LIN {X 0,Y 496.767,Z 453.608,A -85,B 0,C 180,E1 23581.384,E2 23581.384} C_VEL
LIN {X 0,Y 496.758,Z 453.609,A -85,B 0,C 180,E1 23577.924,E2 23577.924} C_VEL
LIN {X 0,Y 496.728,Z 453.609,A -85,B 0,C 180,E1 23574.339,E2 23574.339} C_VEL
LIN {X 0,Y 496.766,Z 453.603,A -85,B 0,C 180,E1 23570.967,E2 23570.967} C_VEL
LIN {X 0,Y 496.72,Z 453.602,A -85,B 0,C 180,E1 23567.444,E2 23567.444} C_VEL
LIN {X 0,Y 496.743,Z 453.608,A -85,B 0,C 180,E1 23563.753,E2 23563.753} C_VEL
LIN {X 0,Y 496.771,Z 453.603,A -85,B 0,C 180,E1 23560.236,E2 23560.236} C_VEL
LIN {X 0,Y 496.761,Z 453.6,A -85,B 0,C 180,E1 23556.607,E2 23556.607} C_VEL
LIN {X 0,Y 496.76,Z 453.601,A -85,B 0,C 180,E1 23553.072,E2 23553.072} C_VEL
LIN {X 0,Y 496.74,Z 453.605,A -85,B 0,C 180,E1 23549.654,E2 23549.654} C_VEL
LIN {X 0,Y 496.768,Z 453.604,A -85,B 0,C 180,E1 23546.227,E2 23546.227} C_VEL
LIN {X 0,Y 496.727,Z 453.608,A -85,B 0,C 180,E1 23542.663,E2 23542.663} C_VEL
LIN {X 0,Y 496.74,Z 453.603,A -85,B 0,C 180,E1 23538.99,E2 23538.99} C_VEL
LIN {X 0,Y 496.772,Z 453.607,A -85,B 0,C 180,E1 23535.438,E2 23535.438} C_VEL
LIN {X 0,Y 496.756,Z 453.607,A -85,B 0,C 180,E1 23531.776,E2 23531.776} C_VEL
LIN {X 0,Y 496.797,Z 453.816,A -85,B 0,C 180,E1 23528.426,E2 23528.426} C_VEL
LIN {X 0,Y 499.428,Z 460.561,A -85,B 0,C 180,E1 23527.574,E2 23527.574} C_VEL
LIN {X 0,Y 500.967,Z 466.815,A -85,B 0,C 180,E1 23526.871,E2 23526.871} C_VEL
LIN {X 0,Y 501.424,Z 476.32,A -85,B 0,C 180,E1 23525.981,E2 23525.981} C_VEL
LIN {X 0,Y 500.918,Z 488.092,A -85,B 0,C 180,E1 23524.986,E2 23524.986} C_VEL
LIN {X 0,Y 500.767,Z 497.539,A -85,B 0,C 180,E1 23524.262,E2 23524.262} C_VEL
LIN {X 0,Y 504.297,Z 517.076,A -85,B 0,C 180,E1 23523.658,E2 23523.658} C_VEL
LIN {X 0,Y 500.785,Z 757.312,A -85,B 0,C 180,E1 23519.902,E2 23519.902} C_VEL
LIN {X 0,Y 500.061,Z 778.117,A -85,B 0,C 180,E1 23519.377,E2 23519.377} C_VEL
LIN {X 0,Y 499.115,Z 798.423,A -85,B 0,C 180,E1 23518.641,E2 23518.641} C_VEL
LIN {X 0,Y 498.011,Z 817.074,A -85,B 0,C 180,E1 23517.76,E2 23517.76} C_VEL
LIN {X 0,Y 496.743,Z 835.707,A -85,B 0,C 180,E1 23516.658,E2 23516.658} C_VEL
LIN {X 0,Y 495.333,Z 853.877,A -85,B 0,C 180,E1 23515.336,E2 23515.336} C_VEL
LIN {X 0,Y 493.958,Z 870.504,A -85,B 0,C 180,E1 23513.88,E2 23513.88} C_VEL
LIN {X 0,Y 492.63,Z 886.184,A -85,B 0,C 180,E1 23512.254,E2 23512.254} C_VEL
LIN {X 0,Y 491.341,Z 901.557,A -85,B 0,C 180,E1 23510.363,E2 23510.363} C_VEL
LIN {X 0,Y 490.291,Z 914.845,A -85,B 0,C 180,E1 23508.426,E2 23508.426} C_VEL
LIN {X 0,Y 489.403,Z 927.72,A -85,B 0,C 180,E1 23506.215,E2 23506.215} C_VEL
LIN {X 0,Y 488.799,Z 938.134,A -85,B 0,C 180,E1 23504.088,E2 23504.088} C_VEL
LIN {X 0,Y 488.371,Z 947.278,A -85,B 0,C 180,E1 23501.813,E2 23501.813} C_VEL
LIN {X 0,Y 488.112,Z 954.541,A -85,B 0,C 180,E1 23499.55,E2 23499.55} C_VEL
LIN {X 0,Y 487.969,Z 960.402,A -85,B 0,C 180,E1 23497.18,E2 23497.18} C_VEL
LIN {X 0,Y 487.924,Z 964.548,A -85,B 0,C 180,E1 23494.819,E2 23494.819} C_VEL
LIN {X 0,Y 487.91,Z 967.076,A -85,B 0,C 180,E1 23492.466,E2 23492.466} C_VEL
LIN {X 0,Y 487.913,Z 967.976,A -85,B 0,C 180,E1 23490.117,E2 23490.117} C_VEL
LIN {X 0,Y 487.909,Z 967.263,A -85,B 0,C 180,E1 23487.768,E2 23487.768} C_VEL
LIN {X 0,Y 487.924,Z 964.827,A -85,B 0,C 180,E1 23485.298,E2 23485.298} C_VEL
LIN {X 0,Y 487.969,Z 960.841,A -85,B 0,C 180,E1 23482.937,E2 23482.937} C_VEL
LIN {X 0,Y 488.083,Z 955.495,A -85,B 0,C 180,E1 23480.686,E2 23480.686} C_VEL
LIN {X 0,Y 488.341,Z 948.011,A -85,B 0,C 180,E1 23478.305,E2 23478.305} C_VEL
LIN {X 0,Y 488.752,Z 939.018,A -85,B 0,C 180,E1 23476.03,E2 23476.03} C_VEL
LIN {X 0,Y 489.344,Z 928.607,A -85,B 0,C 180,E1 23473.865,E2 23473.865} C_VEL
LIN {X 0,Y 490.248,Z 915.382,A -85,B 0,C 180,E1 23471.571,E2 23471.571} C_VEL
LIN {X 0,Y 491.291,Z 902.2,A -85,B 0,C 180,E1 23469.633,E2 23469.633} C_VEL
LIN {X 0,Y 492.55,Z 887.185,A -85,B 0,C 180,E1 23467.769,E2 23467.769} C_VEL
LIN {X 0,Y 493.883,Z 871.412,A -85,B 0,C 180,E1 23466.115,E2 23466.115} C_VEL
LIN {X 0,Y 495.259,Z 854.963,A -85,B 0,C 180,E1 23464.659,E2 23464.659} C_VEL
LIN {X 0,Y 496.656,Z 836.769,A -85,B 0,C 180,E1 23463.324,E2 23463.324} C_VEL
LIN {X 0,Y 497.902,Z 818.576,A -85,B 0,C 180,E1 23462.232,E2 23462.232} C_VEL
LIN {X 0,Y 499.046,Z 799.72,A -85,B 0,C 180,E1 23461.324,E2 23461.324} C_VEL
LIN {X 0,Y 500.002,Z 779.545,A -85,B 0,C 180,E1 23460.577,E2 23460.577} C_VEL
LIN {X 0,Y 500.746,Z 759.184,A -85,B 0,C 180,E1 23460.045,E2 23460.045} C_VEL
LIN {X 0,Y 501.476,Z 712.817,A -85,B 0,C 180,E1 23459.295,E2 23459.295} C_VEL
LIN {X 0,Y 504.071,Z 522.8,A -85,B 0,C 180,E1 23456.331,E2 23456.331} C_VEL
LIN {X 0,Y 497.624,Z 499.033,A -85,B 0,C 180,E1 23455.392,E2 23455.392} C_VEL
LIN {X 0,Y 498.151,Z 484.204,A -85,B 0,C 180,E1 23453.55,E2 23453.55} C_VEL
LIN {X 0,Y 493.227,Z 467.983,A -85,B 0,C 180,E1 23450.916,E2 23450.916} C_VEL
LIN {X 0,Y 488.834,Z 454.598,A -85,B 0,C 180,E1 23448.648,E2 23448.648} C_VEL
LIN {X 0,Y 488.83,Z 454.596,A -85,B 0,C 180,E1 23445.049,E2 23445.049} C_VEL
LIN {X 0,Y 488.816,Z 454.593,A -85,B 0,C 180,E1 23441.509,E2 23441.509} C_VEL
LIN {X 0,Y 488.818,Z 454.597,A -85,B 0,C 180,E1 23437.853,E2 23437.853} C_VEL
LIN {X 0,Y 488.827,Z 454.6,A -85,B 0,C 180,E1 23434.228,E2 23434.228} C_VEL
LIN {X 0,Y 488.837,Z 454.703,A -85,B 0,C 180,E1 23433.789,E2 23433.789} C_VEL
LIN {X 0,Y 496.868,Z 477.285,A -85,B 0,C 180,E1 23430.605,E2 23430.605} C_VEL
LIN {X 0,Y 499.503,Z 486.007,A -85,B 0,C 180,E1 23429.454,E2 23429.454} C_VEL
LIN {X 0,Y 497.948,Z 517.033,A -85,B 0,C 180,E1 23426.28,E2 23426.28} C_VEL
LIN {X 0,Y 496.294,Z 552.146,A -85,B 0,C 180,E1 23422.757,E2 23422.757} C_VEL
LIN {X 0,Y 494.808,Z 586.796,A -85,B 0,C 180,E1 23419.321,E2 23419.321} C_VEL
LIN {X 0,Y 493.925,Z 612.077,A -85,B 0,C 180,E1 23416.881,E2 23416.881} C_VEL
LIN {X 0,Y 494.597,Z 617.905,A -85,B 0,C 180,E1 23416.743,E2 23416.743} C_VEL
LIN {X 0,Y 492.505,Z 754.45,A -85,B 0,C 180,E1 23414.363,E2 23414.363} C_VEL
LIN {X 0,Y 492.275,Z 770.709,A -85,B 0,C 180,E1 23413.862,E2 23413.862} C_VEL
LIN {X 0,Y 491.901,Z 786.257,A -85,B 0,C 180,E1 23413.159,E2 23413.159} C_VEL
LIN {X 0,Y 491.414,Z 801.692,A -85,B 0,C 180,E1 23412.217,E2 23412.217} C_VEL
LIN {X 0,Y 490.893,Z 815.138,A -85,B 0,C 180,E1 23411.157,E2 23411.157} C_VEL
LIN {X 0,Y 490.328,Z 828.203,A -85,B 0,C 180,E1 23409.863,E2 23409.863} C_VEL
LIN {X 0,Y 489.819,Z 839.61,A -85,B 0,C 180,E1 23408.452,E2 23408.452} C_VEL
LIN {X 0,Y 489.359,Z 850.195,A -85,B 0,C 180,E1 23406.806,E2 23406.806} C_VEL
LIN {X 0,Y 489.026,Z 858.519,A -85,B 0,C 180,E1 23405.162,E2 23405.162} C_VEL
LIN {X 0,Y 488.773,Z 865.789,A -85,B 0,C 180,E1 23403.284,E2 23403.284} C_VEL
LIN {X 0,Y 488.622,Z 870.731,A -85,B 0,C 180,E1 23401.525,E2 23401.525} C_VEL
LIN {X 0,Y 488.556,Z 874.365,A -85,B 0,C 180,E1 23399.531,E2 23399.531} C_VEL
LIN {X 0,Y 488.537,Z 876.042,A -85,B 0,C 180,E1 23397.654,E2 23397.654} C_VEL
LIN {X 0,Y 488.584,Z 875.958,A -85,B 0,C 180,E1 23395.658,E2 23395.658} C_VEL
LIN {X 0,Y 488.669,Z 874.165,A -85,B 0,C 180,E1 23393.775,E2 23393.775} C_VEL
LIN {X 0,Y 488.857,Z 870.319,A -85,B 0,C 180,E1 23391.769,E2 23391.769} C_VEL
LIN {X 0,Y 489.105,Z 865.112,A -85,B 0,C 180,E1 23389.994,E2 23389.994} C_VEL
LIN {X 0,Y 489.458,Z 857.991,A -85,B 0,C 180,E1 23388.213,E2 23388.213} C_VEL
LIN {X 0,Y 489.875,Z 849.994,A -85,B 0,C 180,E1 23386.666,E2 23386.666} C_VEL
LIN {X 0,Y 490.403,Z 839.836,A -85,B 0,C 180,E1 23385.111,E2 23385.111} C_VEL
LIN {X 0,Y 490.983,Z 828.633,A -85,B 0,C 180,E1 23383.739,E2 23383.739} C_VEL
LIN {X 0,Y 491.568,Z 815.645,A -85,B 0,C 180,E1 23382.48,E2 23382.48} C_VEL
LIN {X 0,Y 492.065,Z 802.422,A -85,B 0,C 180,E1 23381.466,E2 23381.466} C_VEL
LIN {X 0,Y 492.467,Z 787.433,A -85,B 0,C 180,E1 23380.587,E2 23380.587} C_VEL
LIN {X 0,Y 492.728,Z 772.16,A -85,B 0,C 180,E1 23379.93,E2 23379.93} C_VEL
LIN {X 0,Y 492.8,Z 755.484,A -85,B 0,C 180,E1 23379.463,E2 23379.463} C_VEL
LIN {X 0,Y 494.568,Z 679.992,A -85,B 0,C 180,E1 23377.943,E2 23377.943} C_VEL
LIN {X 0,Y 496.475,Z 627.67,A -85,B 0,C 180,E1 23376.814,E2 23376.814} C_VEL
LIN {X 0,Y 499.112,Z 620.24,A -85,B 0,C 180,E1 23376.193,E2 23376.193} C_VEL
LIN {X 0,Y 502.985,Z 587.434,A -85,B 0,C 180,E1 23372.448,E2 23372.448} C_VEL
LIN {X 0,Y 508.02,Z 558.234,A -85,B 0,C 180,E1 23368.888,E2 23368.888} C_VEL
LIN {X 0,Y 513.627,Z 535.581,A -85,B 0,C 180,E1 23365.9,E2 23365.9} C_VEL
LIN {X 0,Y 518.825,Z 520.705,A -85,B 0,C 180,E1 23363.727,E2 23363.727} C_VEL
LIN {X 0,Y 521.042,Z 515.3,A -85,B 0,C 180,E1 23362.786,E2 23362.786} C_VEL
LIN {X 0,Y 521.265,Z 512.97,A -85,B 0,C 180,E1 23361.5,E2 23361.5} C_VEL
LIN {X 0,Y 521.568,Z 512.33,A -85,B 0,C 180,E1 23360.757,E2 23360.757} C_VEL
LIN {X 0,Y 521.764,Z 512.428,A -85,B 0,C 180,E1 23360.176,E2 23360.176} C_VEL
LIN {X 0,Y 514.97,Z 524.97,A -85,B 0,C 180,E1 23358.69,E2 23358.69} C_VEL
LIN {X 0,Y 509.541,Z 539.534,A -85,B 0,C 180,E1 23357.132,E2 23357.132} C_VEL
LIN {X 0,Y 505.219,Z 557.552,A -85,B 0,C 180,E1 23355.367,E2 23355.367} C_VEL
LIN {X 0,Y 503.453,Z 574.846,A -85,B 0,C 180,E1 23353.705,E2 23353.705} C_VEL
LIN {X 0,Y 503.998,Z 589.634,A -85,B 0,C 180,E1 23352.263,E2 23352.263} C_VEL
LIN {X 0,Y 506.627,Z 603.149,A -85,B 0,C 180,E1 23350.899,E2 23350.899} C_VEL
LIN {X 0,Y 511.168,Z 615.366,A -85,B 0,C 180,E1 23349.619,E2 23349.619} C_VEL
LIN {X 0,Y 517.239,Z 625.827,A -85,B 0,C 180,E1 23348.474,E2 23348.474} C_VEL
LIN {X 0,Y 524.902,Z 635.189,A -85,B 0,C 180,E1 23347.409,E2 23347.409} C_VEL
LIN {X 0,Y 534.249,Z 643.624,A -85,B 0,C 180,E1 23346.414,E2 23346.414} C_VEL
LIN {X 0,Y 545.236,Z 650.974,A -85,B 0,C 180,E1 23345.491,E2 23345.491} C_VEL
LIN {X 0,Y 557.413,Z 656.852,A -85,B 0,C 180,E1 23344.655,E2 23344.655} C_VEL
LIN {X 0,Y 543.385,Z 678.868,A -85,B 0,C 180,E1 23343.886,E2 23343.886} C_VEL
LIN {X 0,Y 536.689,Z 691.188,A -85,B 0,C 180,E1 23343.397,E2 23343.397} C_VEL
LIN {X 0,Y 523.96,Z 709.583,A -85,B 0,C 180,E1 23342.752,E2 23342.752} C_VEL
LIN {X 0,Y 515.235,Z 724.92,A -85,B 0,C 180,E1 23342.123,E2 23342.123} C_VEL
LIN {X 0,Y 509.382,Z 738.59,A -85,B 0,C 180,E1 23341.476,E2 23341.476} C_VEL
LIN {X 0,Y 502.738,Z 756.016,A -85,B 0,C 180,E1 23340.607,E2 23340.607} C_VEL
LIN {X 0,Y 501.2,Z 761.517,A -85,B 0,C 180,E1 23340.344,E2 23340.344} C_VEL
LIN {X 0,Y 500.102,Z 775.893,A -85,B 0,C 180,E1 23340.184,E2 23340.184} C_VEL
LIN {X 0,Y 499.546,Z 807.756,A -85,B 0,C 180,E1 23339.646,E2 23339.646} C_VEL
LIN {X 0,Y 498.768,Z 828.234,A -85,B 0,C 180,E1 23339.099,E2 23339.099} C_VEL
LIN {X 0,Y 497.811,Z 848.512,A -85,B 0,C 180,E1 23338.331,E2 23338.331} C_VEL
LIN {X 0,Y 496.699,Z 867.553,A -85,B 0,C 180,E1 23337.393,E2 23337.393} C_VEL
LIN {X 0,Y 495.441,Z 886.583,A -85,B 0,C 180,E1 23336.23,E2 23336.23} C_VEL
LIN {X 0,Y 494.152,Z 905.345,A -85,B 0,C 180,E1 23334.826,E2 23334.826} C_VEL
LIN {X 0,Y 492.687,Z 927.463,A -85,B 0,C 180,E1 23332.877,E2 23332.877} C_VEL
LIN {X 0,Y 491.821,Z 940.657,A -85,B 0,C 180,E1 23331.528,E2 23331.528} C_VEL
LIN {X 0,Y 490.937,Z 954.693,A -85,B 0,C 180,E1 23329.885,E2 23329.885} C_VEL
LIN {X 0,Y 490.153,Z 966.564,A -85,B 0,C 180,E1 23328.187,E2 23328.187} C_VEL
LIN {X 0,Y 489.434,Z 977.053,A -85,B 0,C 180,E1 23326.375,E2 23326.375} C_VEL
LIN {X 0,Y 488.843,Z 987.247,A -85,B 0,C 180,E1 23324.33,E2 23324.33} C_VEL
LIN {X 0,Y 488.409,Z 996.057,A -85,B 0,C 180,E1 23322.173,E2 23322.173} C_VEL
LIN {X 0,Y 488.147,Z 1003.268,A -85,B 0,C 180,E1 23320.027,E2 23320.027} C_VEL
LIN {X 0,Y 487.983,Z 1009.716,A -85,B 0,C 180,E1 23317.536,E2 23317.536} C_VEL
LIN {X 0,Y 487.926,Z 1013.53,A -85,B 0,C 180,E1 23315.527,E2 23315.527} C_VEL
LIN {X 0,Y 487.905,Z 1016.55,A -85,B 0,C 180,E1 23313.172,E2 23313.172} C_VEL
LIN {X 0,Y 487.908,Z 1017.826,A -85,B 0,C 180,E1 23310.823,E2 23310.823} C_VEL
LIN {X 0,Y 487.9,Z 1017.687,A -85,B 0,C 180,E1 23308.591,E2 23308.591} C_VEL
LIN {X 0,Y 487.916,Z 1015.774,A -85,B 0,C 180,E1 23306.123,E2 23306.123} C_VEL
LIN {X 0,Y 487.948,Z 1012.753,A -85,B 0,C 180,E1 23304.002,E2 23304.002} C_VEL
LIN {X 0,Y 488.044,Z 1007.51,A -85,B 0,C 180,E1 23301.518,E2 23301.518} C_VEL
LIN {X 0,Y 488.21,Z 1001.413,A -85,B 0,C 180,E1 23299.379,E2 23299.379} C_VEL
LIN {X 0,Y 488.548,Z 993.366,A -85,B 0,C 180,E1 23297.111,E2 23297.111} C_VEL
LIN {X 0,Y 489.023,Z 983.808,A -85,B 0,C 180,E1 23294.95,E2 23294.95} C_VEL
LIN {X 0,Y 489.733,Z 972.785,A -85,B 0,C 180,E1 23292.84,E2 23292.84} C_VEL
LIN {X 0,Y 490.482,Z 961.579,A -85,B 0,C 180,E1 23291.062,E2 23291.062} C_VEL
LIN {X 0,Y 491.252,Z 949.885,A -85,B 0,C 180,E1 23289.509,E2 23289.509} C_VEL
LIN {X 0,Y 492.326,Z 934.537,A -85,B 0,C 180,E1 23287.744,E2 23287.744} C_VEL
LIN {X 0,Y 493.5,Z 917.544,A -85,B 0,C 180,E1 23286.096,E2 23286.096} C_VEL
LIN {X 0,Y 494.712,Z 899.66,A -85,B 0,C 180,E1 23284.63,E2 23284.63} C_VEL
LIN {X 0,Y 496.011,Z 879.286,A -85,B 0,C 180,E1 23283.252,E2 23283.252} C_VEL
LIN {X 0,Y 497.185,Z 860.173,A -85,B 0,C 180,E1 23282.189,E2 23282.189} C_VEL
LIN {X 0,Y 498.27,Z 839.247,A -85,B 0,C 180,E1 23281.272,E2 23281.272} C_VEL
LIN {X 0,Y 499.25,Z 817.685,A -85,B 0,C 180,E1 23280.564,E2 23280.564} C_VEL
LIN {X 0,Y 499.975,Z 795.148,A -85,B 0,C 180,E1 23280.068,E2 23280.068} C_VEL
LIN {X 0,Y 500.611,Z 768.473,A -85,B 0,C 180,E1 23279.649,E2 23279.649} C_VEL
LIN {X 0,Y 506.326,Z 750.486,A -85,B 0,C 180,E1 23278.712,E2 23278.712} C_VEL
LIN {X 0,Y 510.554,Z 739.866,A -85,B 0,C 180,E1 23278.211,E2 23278.211} C_VEL
LIN {X 0,Y 516.327,Z 726.256,A -85,B 0,C 180,E1 23277.597,E2 23277.597} C_VEL
LIN {X 0,Y 524.549,Z 711.279,A -85,B 0,C 180,E1 23277.037,E2 23277.037} C_VEL
LIN {X 0,Y 537.482,Z 691.726,A -85,B 0,C 180,E1 23276.449,E2 23276.449} C_VEL
LIN {X 0,Y 547.16,Z 673.813,A -85,B 0,C 180,E1 23275.812,E2 23275.812} C_VEL
LIN {X 0,Y 557.517,Z 656.992,A -85,B 0,C 180,E1 23275.302,E2 23275.302} C_VEL
LIN {X 0,Y 546.441,Z 652.277,A -85,B 0,C 180,E1 23274.332,E2 23274.332} C_VEL
LIN {X 0,Y 536.165,Z 645.852,A -85,B 0,C 180,E1 23273.23,E2 23273.23} C_VEL
LIN {X 0,Y 527.366,Z 638.017,A -85,B 0,C 180,E1 23272.065,E2 23272.065} C_VEL
LIN {X 0,Y 520.404,Z 629.287,A -85,B 0,C 180,E1 23270.915,E2 23270.915} C_VEL
LIN {X 0,Y 514.442,Z 618.41,A -85,B 0,C 180,E1 23269.63,E2 23269.63} C_VEL
LIN {X 0,Y 510.166,Z 605.832,A -85,B 0,C 180,E1 23268.306,E2 23268.306} C_VEL
LIN {X 0,Y 507.583,Z 591.714,A -85,B 0,C 180,E1 23266.954,E2 23266.954} C_VEL
LIN {X 0,Y 506.67,Z 574.593,A -85,B 0,C 180,E1 23265.48,E2 23265.48} C_VEL
LIN {X 0,Y 508.228,Z 544.689,A -85,B 0,C 180,E1 23263.124,E2 23263.124} C_VEL
LIN {X 0,Y 510.988,Z 507.421,A -85,B 0,C 180,E1 23260.174,E2 23260.174} C_VEL
LIN {X 0,Y 511.243,Z 500.742,A -85,B 0,C 180,E1 23259.611,E2 23259.611} C_VEL
LIN {X 0,Y 501.377,Z 480.291,A -85,B 0,C 180,E1 23256.603,E2 23256.603} C_VEL
LIN {X 0,Y 492.527,Z 462.708,A -85,B 0,C 180,E1 23253.796,E2 23253.796} C_VEL
LIN {X 0,Y 490.299,Z 458.319,A -85,B 0,C 180,E1 23253.056,E2 23253.056} C_VEL
LIN {X 0,Y 488.898,Z 455.069,A -85,B 0,C 180,E1 23252.538,E2 23252.538} C_VEL
LIN {X 0,Y 488.824,Z 454.586,A -85,B 0,C 180,E1 23252.405,E2 23252.405} C_VEL
LIN {X 0,Y 488.78,Z 454.599,A -85,B 0,C 180,E1 23248.866,E2 23248.866} C_VEL
LIN {X 0,Y 488.812,Z 454.598,A -85,B 0,C 180,E1 23245.18,E2 23245.18} C_VEL
LIN {X 0,Y 488.836,Z 454.595,A -85,B 0,C 180,E1 23241.603,E2 23241.603} C_VEL
LIN {X 0,Y 488.835,Z 454.597,A -85,B 0,C 180,E1 23237.867,E2 23237.867} C_VEL
LIN {X 0,Y 488.81,Z 454.6,A -85,B 0,C 180,E1 23234.33,E2 23234.33} C_VEL
LIN {X 0,Y 488.782,Z 454.601,A -85,B 0,C 180,E1 23230.728,E2 23230.728} C_VEL
LIN {X 0,Y 488.834,Z 454.592,A -85,B 0,C 180,E1 23227.25,E2 23227.25} C_VEL
LIN {X 0,Y 488.781,Z 454.601,A -85,B 0,C 180,E1 23223.753,E2 23223.753} C_VEL
LIN {X 0,Y 488.815,Z 454.595,A -85,B 0,C 180,E1 23220.117,E2 23220.117} C_VEL
LIN {X 0,Y 488.826,Z 454.597,A -85,B 0,C 180,E1 23216.523,E2 23216.523} C_VEL
LIN {X 0,Y 488.83,Z 454.583,A -85,B 0,C 180,E1 23212.754,E2 23212.754} C_VEL
LIN {X 0,Y 488.809,Z 454.596,A -85,B 0,C 180,E1 23209.272,E2 23209.272} C_VEL
LIN {X 0,Y 488.779,Z 454.596,A -85,B 0,C 180,E1 23205.548,E2 23205.548} C_VEL
LIN {X 0,Y 488.825,Z 454.585,A -85,B 0,C 180,E1 23202.009,E2 23202.009} C_VEL
LIN {X 0,Y 488.805,Z 454.598,A -85,B 0,C 180,E1 23198.522,E2 23198.522} C_VEL
LIN {X 0,Y 488.826,Z 454.599,A -85,B 0,C 180,E1 23194.95,E2 23194.95} C_VEL
LIN {X 0,Y 488.812,Z 454.601,A -85,B 0,C 180,E1 23191.403,E2 23191.403} C_VEL
LIN {X 0,Y 488.826,Z 454.597,A -85,B 0,C 180,E1 23187.865,E2 23187.865} C_VEL
LIN {X 0,Y 488.813,Z 454.597,A -85,B 0,C 180,E1 23184.296,E2 23184.296} C_VEL
LIN {X 0,Y 488.78,Z 454.601,A -85,B 0,C 180,E1 23180.643,E2 23180.643} C_VEL
LIN {X 0,Y 488.822,Z 454.597,A -85,B 0,C 180,E1 23177.068,E2 23177.068} C_VEL
LIN {X 0,Y 488.817,Z 454.596,A -85,B 0,C 180,E1 23173.576,E2 23173.576} C_VEL
LIN {X 0,Y 488.826,Z 454.594,A -85,B 0,C 180,E1 23170.094,E2 23170.094} C_VEL
LIN {X 0,Y 488.841,Z 454.721,A -85,B 0,C 180,E1 23169.066,E2 23169.066} C_VEL
LIN {X 0,Y 498.209,Z 478.903,A -85,B 0,C 180,E1 23166.016,E2 23166.016} C_VEL
LIN {X 0,Y 500.967,Z 486.916,A -85,B 0,C 180,E1 23165.085,E2 23165.085} C_VEL
LIN {X 0,Y 500.918,Z 488.092,A -85,B 0,C 180,E1 23164.986,E2 23164.986} C_VEL
LIN {X 0,Y 500.479,Z 493.877,A -85,B 0,C 180,E1 23164.621,E2 23164.621} C_VEL
LIN {X 0,Y 499.47,Z 502.377,A -85,B 0,C 180,E1 23164.345,E2 23164.345} C_VEL
LIN {X 0,Y 497.597,Z 521.582,A -85,B 0,C 180,E1 23164.1,E2 23164.1} C_VEL
LIN {X 0,Y 497.569,Z 522.676,A -85,B 0,C 180,E1 23164.084,E2 23164.084} C_VEL
LIN {X 0,Y 493.861,Z 757.764,A -85,B 0,C 180,E1 23160.36,E2 23160.36} C_VEL
LIN {X 0,Y 493.095,Z 778.615,A -85,B 0,C 180,E1 23159.827,E2 23159.827} C_VEL
LIN {X 0,Y 492.09,Z 798.85,A -85,B 0,C 180,E1 23159.086,E2 23159.086} C_VEL
LIN {X 0,Y 490.921,Z 817.45,A -85,B 0,C 180,E1 23158.197,E2 23158.197} C_VEL
LIN {X 0,Y 489.539,Z 836.369,A -85,B 0,C 180,E1 23157.062,E2 23157.062} C_VEL
LIN {X 0,Y 487.989,Z 855.062,A -85,B 0,C 180,E1 23155.68,E2 23155.68} C_VEL
LIN {X 0,Y 486.449,Z 872.327,A -85,B 0,C 180,E1 23154.131,E2 23154.131} C_VEL
LIN {X 0,Y 485.03,Z 887.772,A -85,B 0,C 180,E1 23152.482,E2 23152.482} C_VEL
LIN {X 0,Y 483.735,Z 901.971,A -85,B 0,C 180,E1 23150.698,E2 23150.698} C_VEL
LIN {X 0,Y 482.588,Z 915.262,A -85,B 0,C 180,E1 23148.731,E2 23148.731} C_VEL
LIN {X 0,Y 481.651,Z 927.161,A -85,B 0,C 180,E1 23146.646,E2 23146.646} C_VEL
LIN {X 0,Y 480.931,Z 937.66,A -85,B 0,C 180,E1 23144.446,E2 23144.446} C_VEL
LIN {X 0,Y 480.417,Z 947.358,A -85,B 0,C 180,E1 23141.99,E2 23141.99} C_VEL
LIN {X 0,Y 480.125,Z 954.892,A -85,B 0,C 180,E1 23139.59,E2 23139.59} C_VEL
LIN {X 0,Y 479.977,Z 960.403,A -85,B 0,C 180,E1 23137.3,E2 23137.3} C_VEL
LIN {X 0,Y 479.924,Z 964.548,A -85,B 0,C 180,E1 23134.899,E2 23134.899} C_VEL
LIN {X 0,Y 479.91,Z 967.076,A -85,B 0,C 180,E1 23132.507,E2 23132.507} C_VEL
LIN {X 0,Y 479.914,Z 967.976,A -85,B 0,C 180,E1 23130.119,E2 23130.119} C_VEL
LIN {X 0,Y 479.909,Z 967.262,A -85,B 0,C 180,E1 23127.731,E2 23127.731} C_VEL
LIN {X 0,Y 479.924,Z 964.984,A -85,B 0,C 180,E1 23125.339,E2 23125.339} C_VEL
LIN {X 0,Y 479.973,Z 961.092,A -85,B 0,C 180,E1 23122.939,E2 23122.939} C_VEL
LIN {X 0,Y 480.105,Z 955.493,A -85,B 0,C 180,E1 23120.53,E2 23120.53} C_VEL
LIN {X 0,Y 480.391,Z 948.008,A -85,B 0,C 180,E1 23118.108,E2 23118.108} C_VEL
LIN {X 0,Y 480.842,Z 939.03,A -85,B 0,C 180,E1 23115.796,E2 23115.796} C_VEL
LIN {X 0,Y 481.523,Z 928.832,A -85,B 0,C 180,E1 23113.596,E2 23113.596} C_VEL
LIN {X 0,Y 482.481,Z 916.537,A -85,B 0,C 180,E1 23111.389,E2 23111.389} C_VEL
LIN {X 0,Y 483.683,Z 902.602,A -85,B 0,C 180,E1 23109.299,E2 23109.299} C_VEL
LIN {X 0,Y 485.014,Z 887.978,A -85,B 0,C 180,E1 23107.452,E2 23107.452} C_VEL
LIN {X 0,Y 486.439,Z 872.45,A -85,B 0,C 180,E1 23105.79,E2 23105.79} C_VEL
LIN {X 0,Y 487.968,Z 855.342,A -85,B 0,C 180,E1 23104.253,E2 23104.253} C_VEL
LIN {X 0,Y 489.472,Z 837.135,A -85,B 0,C 180,E1 23102.9,E2 23102.9} C_VEL
LIN {X 0,Y 490.805,Z 818.924,A -85,B 0,C 180,E1 23101.794,E2 23101.794} C_VEL
LIN {X 0,Y 492.054,Z 799.487,A -85,B 0,C 180,E1 23100.852,E2 23100.852} C_VEL
LIN {X 0,Y 493.09,Z 778.706,A -85,B 0,C 180,E1 23100.085,E2 23100.085} C_VEL
LIN {X 0,Y 493.862,Z 757.779,A -85,B 0,C 180,E1 23099.55,E2 23099.55} C_VEL
LIN {X 0,Y 497.456,Z 524.753,A -85,B 0,C 180,E1 23095.853,E2 23095.853} C_VEL
LIN {X 0,Y 490.54,Z 499.338,A -85,B 0,C 180,E1 23094.821,E2 23094.821} C_VEL
LIN {X 0,Y 490.844,Z 486.961,A -85,B 0,C 180,E1 23093.28,E2 23093.28} C_VEL
LIN {X 0,Y 486.326,Z 471.941,A -85,B 0,C 180,E1 23090.814,E2 23090.814} C_VEL
LIN {X 0,Y 481.43,Z 457.68,A -85,B 0,C 180,E1 23088.348,E2 23088.348} C_VEL
LIN {X 0,Y 480.86,Z 455.591,A -85,B 0,C 180,E1 23087.968,E2 23087.968} C_VEL
LIN {X 0,Y 480.882,Z 455.58,A -85,B 0,C 180,E1 23084.335,E2 23084.335} C_VEL
LIN {X 0,Y 480.887,Z 455.585,A -85,B 0,C 180,E1 23080.758,E2 23080.758} C_VEL
LIN {X 0,Y 480.888,Z 455.588,A -85,B 0,C 180,E1 23077.083,E2 23077.083} C_VEL
LIN {X 0,Y 480.909,Z 455.781,A -85,B 0,C 180,E1 23074.399,E2 23074.399} C_VEL
LIN {X 0,Y 488.622,Z 477.152,A -85,B 0,C 180,E1 23071.316,E2 23071.316} C_VEL
LIN {X 0,Y 492.351,Z 489.049,A -85,B 0,C 180,E1 23069.704,E2 23069.704} C_VEL
LIN {X 0,Y 490.707,Z 520.139,A -85,B 0,C 180,E1 23066.502,E2 23066.502} C_VEL
LIN {X 0,Y 488.876,Z 555.998,A -85,B 0,C 180,E1 23062.867,E2 23062.867} C_VEL
LIN {X 0,Y 487.33,Z 591.228,A -85,B 0,C 180,E1 23059.351,E2 23059.351} C_VEL
LIN {X 0,Y 486.516,Z 613.109,A -85,B 0,C 180,E1 23057.228,E2 23057.228} C_VEL
LIN {X 0,Y 487.182,Z 618.985,A -85,B 0,C 180,E1 23057.082,E2 23057.082} C_VEL
LIN {X 0,Y 484.883,Z 755.648,A -85,B 0,C 180,E1 23054.628,E2 23054.628} C_VEL
LIN {X 0,Y 484.63,Z 772.532,A -85,B 0,C 180,E1 23054.09,E2 23054.09} C_VEL
LIN {X 0,Y 484.226,Z 787.918,A -85,B 0,C 180,E1 23053.372,E2 23053.372} C_VEL
LIN {X 0,Y 483.712,Z 803.212,A -85,B 0,C 180,E1 23052.414,E2 23052.414} C_VEL
LIN {X 0,Y 483.158,Z 816.554,A -85,B 0,C 180,E1 23051.338,E2 23051.338} C_VEL
LIN {X 0,Y 482.557,Z 829.574,A -85,B 0,C 180,E1 23050.023,E2 23050.023} C_VEL
LIN {X 0,Y 482.015,Z 840.935,A -85,B 0,C 180,E1 23048.59,E2 23048.59} C_VEL
LIN {X 0,Y 481.524,Z 851.51,A -85,B 0,C 180,E1 23046.917,E2 23046.917} C_VEL
LIN {X 0,Y 481.163,Z 859.812,A -85,B 0,C 180,E1 23045.246,E2 23045.246} C_VEL
LIN {X 0,Y 480.891,Z 867.088,A -85,B 0,C 180,E1 23043.338,E2 23043.338} C_VEL
LIN {X 0,Y 480.726,Z 872.015,A -85,B 0,C 180,E1 23041.55,E2 23041.55} C_VEL
LIN {X 0,Y 480.657,Z 875.659,A -85,B 0,C 180,E1 23039.523,E2 23039.523} C_VEL
LIN {X 0,Y 480.637,Z 877.317,A -85,B 0,C 180,E1 23037.616,E2 23037.616} C_VEL
LIN {X 0,Y 480.695,Z 877.239,A -85,B 0,C 180,E1 23035.586,E2 23035.586} C_VEL
LIN {X 0,Y 480.791,Z 875.411,A -85,B 0,C 180,E1 23033.672,E2 23033.672} C_VEL
LIN {X 0,Y 481.01,Z 871.561,A -85,B 0,C 180,E1 23031.634,E2 23031.634} C_VEL
LIN {X 0,Y 481.289,Z 866.319,A -85,B 0,C 180,E1 23029.829,E2 23029.829} C_VEL
LIN {X 0,Y 481.694,Z 859.203,A -85,B 0,C 180,E1 23028.02,E2 23028.02} C_VEL
LIN {X 0,Y 482.154,Z 851.171,A -85,B 0,C 180,E1 23026.448,E2 23026.448} C_VEL
LIN {X 0,Y 482.756,Z 840.739,A -85,B 0,C 180,E1 23024.833,E2 23024.833} C_VEL
LIN {X 0,Y 483.363,Z 829.693,A -85,B 0,C 180,E1 23023.476,E2 23023.476} C_VEL
LIN {X 0,Y 484.003,Z 816.691,A -85,B 0,C 180,E1 23022.198,E2 23022.198} C_VEL
LIN {X 0,Y 484.544,Z 803.092,A -85,B 0,C 180,E1 23021.149,E2 23021.149} C_VEL
LIN {X 0,Y 484.963,Z 788.926,A -85,B 0,C 180,E1 23020.304,E2 23020.304} C_VEL
LIN {X 0,Y 485.233,Z 773.911,A -85,B 0,C 180,E1 23019.648,E2 23019.648} C_VEL
LIN {X 0,Y 485.306,Z 757.393,A -85,B 0,C 180,E1 23019.171,E2 23019.171} C_VEL
LIN {X 0,Y 487.184,Z 685.998,A -85,B 0,C 180,E1 23017.659,E2 23017.659} C_VEL
LIN {X 0,Y 489.477,Z 630.478,A -85,B 0,C 180,E1 23016.399,E2 23016.399} C_VEL
LIN {X 0,Y 492.509,Z 622.313,A -85,B 0,C 180,E1 23015.719,E2 23015.719} C_VEL
LIN {X 0,Y 496.657,Z 590.668,A -85,B 0,C 180,E1 23012.026,E2 23012.026} C_VEL
LIN {X 0,Y 501.97,Z 562.757,A -85,B 0,C 180,E1 23008.542,E2 23008.542} C_VEL
LIN {X 0,Y 507.951,Z 540.77,A -85,B 0,C 180,E1 23005.566,E2 23005.566} C_VEL
LIN {X 0,Y 513.879,Z 525.614,A -85,B 0,C 180,E1 23003.287,E2 23003.287} C_VEL
LIN {X 0,Y 516.053,Z 521.003,A -85,B 0,C 180,E1 23002.458,E2 23002.458} C_VEL
LIN {X 0,Y 516.714,Z 518.751,A -85,B 0,C 180,E1 23000.89,E2 23000.89} C_VEL
LIN {X 0,Y 516.731,Z 518.835,A -85,B 0,C 180,E1 23000.54,E2 23000.54} C_VEL
LIN {X 0,Y 509.623,Z 531.018,A -85,B 0,C 180,E1 22999.057,E2 22999.057} C_VEL
LIN {X 0,Y 503.816,Z 545.093,A -85,B 0,C 180,E1 22997.5,E2 22997.5} C_VEL
LIN {X 0,Y 499.32,Z 561.695,A -85,B 0,C 180,E1 22995.798,E2 22995.798} C_VEL
LIN {X 0,Y 497.201,Z 578.63,A -85,B 0,C 180,E1 22994.092,E2 22994.092} C_VEL
LIN {X 0,Y 497.455,Z 592.881,A -85,B 0,C 180,E1 22992.638,E2 22992.638} C_VEL
LIN {X 0,Y 499.806,Z 606.352,A -85,B 0,C 180,E1 22991.22,E2 22991.22} C_VEL
LIN {X 0,Y 503.929,Z 618.274,A -85,B 0,C 180,E1 22989.927,E2 22989.927} C_VEL
LIN {X 0,Y 509.895,Z 629.189,A -85,B 0,C 180,E1 22988.699,E2 22988.699} C_VEL
LIN {X 0,Y 517.3,Z 638.757,A -85,B 0,C 180,E1 22987.584,E2 22987.584} C_VEL
LIN {X 0,Y 526.394,Z 647.474,A -85,B 0,C 180,E1 22986.538,E2 22986.538} C_VEL
LIN {X 0,Y 537.962,Z 655.703,A -85,B 0,C 180,E1 22985.505,E2 22985.505} C_VEL
LIN {X 0,Y 546.692,Z 660.631,A -85,B 0,C 180,E1 22984.852,E2 22984.852} C_VEL
LIN {X 0,Y 534.991,Z 679.586,A -85,B 0,C 180,E1 22984.168,E2 22984.168} C_VEL
LIN {X 0,Y 530.11,Z 688.583,A -85,B 0,C 180,E1 22983.809,E2 22983.809} C_VEL
LIN {X 0,Y 517.071,Z 707.472,A -85,B 0,C 180,E1 22983.145,E2 22983.145} C_VEL
LIN {X 0,Y 508.534,Z 722.475,A -85,B 0,C 180,E1 22982.531,E2 22982.531} C_VEL
LIN {X 0,Y 502.543,Z 736.156,A -85,B 0,C 180,E1 22981.887,E2 22981.887} C_VEL
LIN {X 0,Y 495.237,Z 755.358,A -85,B 0,C 180,E1 22980.92,E2 22980.92} C_VEL
LIN {X 0,Y 494.734,Z 757.667,A -85,B 0,C 180,E1 22980.845,E2 22980.845} C_VEL
LIN {X 0,Y 493.205,Z 774.336,A -85,B 0,C 180,E1 22980.674,E2 22980.674} C_VEL
LIN {X 0,Y 492.595,Z 807.117,A -85,B 0,C 180,E1 22980.117,E2 22980.117} C_VEL
LIN {X 0,Y 491.759,Z 827.597,A -85,B 0,C 180,E1 22979.567,E2 22979.567} C_VEL
LIN {X 0,Y 490.698,Z 848.043,A -85,B 0,C 180,E1 22978.786,E2 22978.786} C_VEL
LIN {X 0,Y 489.462,Z 867.605,A -85,B 0,C 180,E1 22977.808,E2 22977.808} C_VEL
LIN {X 0,Y 488.127,Z 886.158,A -85,B 0,C 180,E1 22976.654,E2 22976.654} C_VEL
LIN {X 0,Y 486.704,Z 904.918,A -85,B 0,C 180,E1 22975.232,E2 22975.232} C_VEL
LIN {X 0,Y 485.287,Z 922.584,A -85,B 0,C 180,E1 22973.625,E2 22973.625} C_VEL
LIN {X 0,Y 484.089,Z 937.99,A -85,B 0,C 180,E1 22971.954,E2 22971.954} C_VEL
LIN {X 0,Y 482.849,Z 956.276,A -85,B 0,C 180,E1 22969.727,E2 22969.727} C_VEL
LIN {X 0,Y 482.056,Z 968.267,A -85,B 0,C 180,E1 22968.003,E2 22968.003} C_VEL
LIN {X 0,Y 481.434,Z 978.639,A -85,B 0,C 180,E1 22966.283,E2 22966.283} C_VEL
LIN {X 0,Y 480.85,Z 988.818,A -85,B 0,C 180,E1 22964.204,E2 22964.204} C_VEL
LIN {X 0,Y 480.426,Z 996.922,A -85,B 0,C 180,E1 22962.135,E2 22962.135} C_VEL
LIN {X 0,Y 480.146,Z 1004.368,A -85,B 0,C 180,E1 22959.833,E2 22959.833} C_VEL
LIN {X 0,Y 479.987,Z 1009.965,A -85,B 0,C 180,E1 22957.542,E2 22957.542} C_VEL
LIN {X 0,Y 479.926,Z 1013.719,A -85,B 0,C 180,E1 22955.5,E2 22955.5} C_VEL
LIN {X 0,Y 479.908,Z 1016.722,A -85,B 0,C 180,E1 22952.986,E2 22952.986} C_VEL
LIN {X 0,Y 479.905,Z 1017.851,A -85,B 0,C 180,E1 22950.717,E2 22950.717} C_VEL
LIN {X 0,Y 479.903,Z 1017.61,A -85,B 0,C 180,E1 22948.329,E2 22948.329} C_VEL
LIN {X 0,Y 479.92,Z 1015.631,A -85,B 0,C 180,E1 22945.939,E2 22945.939} C_VEL
LIN {X 0,Y 479.955,Z 1012.554,A -85,B 0,C 180,E1 22943.782,E2 22943.782} C_VEL
LIN {X 0,Y 480.065,Z 1007.194,A -85,B 0,C 180,E1 22941.255,E2 22941.255} C_VEL
LIN {X 0,Y 480.244,Z 1001.407,A -85,B 0,C 180,E1 22939.201,E2 22939.201} C_VEL
LIN {X 0,Y 480.616,Z 993.361,A -85,B 0,C 180,E1 22936.894,E2 22936.894} C_VEL
LIN {X 0,Y 481.069,Z 984.911,A -85,B 0,C 180,E1 22934.942,E2 22934.942} C_VEL
LIN {X 0,Y 481.551,Z 976.586,A -85,B 0,C 180,E1 22933.35,E2 22933.35} C_VEL
LIN {X 0,Y 482.345,Z 964.638,A -85,B 0,C 180,E1 22931.384,E2 22931.384} C_VEL
LIN {X 0,Y 483.31,Z 950.347,A -85,B 0,C 180,E1 22929.41,E2 22929.41} C_VEL
LIN {X 0,Y 484.353,Z 936.271,A -85,B 0,C 180,E1 22927.735,E2 22927.735} C_VEL
LIN {X 0,Y 485.603,Z 919.168,A -85,B 0,C 180,E1 22926.006,E2 22926.006} C_VEL
LIN {X 0,Y 487.129,Z 898.952,A -85,B 0,C 180,E1 22924.278,E2 22924.278} C_VEL
LIN {X 0,Y 488.192,Z 884.182,A -85,B 0,C 180,E1 22923.22,E2 22923.22} C_VEL
LIN {X 0,Y 489.411,Z 867.477,A -85,B 0,C 180,E1 22922.179,E2 22922.179} C_VEL
LIN {X 0,Y 490.669,Z 847.563,A -85,B 0,C 180,E1 22921.191,E2 22921.191} C_VEL
LIN {X 0,Y 491.736,Z 826.996,A -85,B 0,C 180,E1 22920.409,E2 22920.409} C_VEL
LIN {X 0,Y 492.564,Z 806.192,A -85,B 0,C 180,E1 22919.857,E2 22919.857} C_VEL
LIN {X 0,Y 493.523,Z 767.721,A -85,B 0,C 180,E1 22919.225,E2 22919.225} C_VEL
LIN {X 0,Y 499.267,Z 749.862,A -85,B 0,C 180,E1 22918.286,E2 22918.286} C_VEL
LIN {X 0,Y 503.852,Z 738.426,A -85,B 0,C 180,E1 22917.737,E2 22917.737} C_VEL
LIN {X 0,Y 509.918,Z 724.422,A -85,B 0,C 180,E1 22917.103,E2 22917.103} C_VEL
LIN {X 0,Y 518.455,Z 708.987,A -85,B 0,C 180,E1 22916.527,E2 22916.527} C_VEL
LIN {X 0,Y 532.271,Z 687.919,A -85,B 0,C 180,E1 22915.895,E2 22915.895} C_VEL
LIN {X 0,Y 540.115,Z 673.279,A -85,B 0,C 180,E1 22915.368,E2 22915.368} C_VEL
LIN {X 0,Y 547.328,Z 661.245,A -85,B 0,C 180,E1 22914.99,E2 22914.99} C_VEL
LIN {X 0,Y 536.673,Z 655.743,A -85,B 0,C 180,E1 22913.956,E2 22913.956} C_VEL
LIN {X 0,Y 527.049,Z 648.767,A -85,B 0,C 180,E1 22912.823,E2 22912.823} C_VEL
LIN {X 0,Y 518.333,Z 639.864,A -85,B 0,C 180,E1 22911.551,E2 22911.551} C_VEL
LIN {X 0,Y 511.406,Z 629.707,A -85,B 0,C 180,E1 22910.259,E2 22910.259} C_VEL
LIN {X 0,Y 506.229,Z 618.507,A -85,B 0,C 180,E1 22908.981,E2 22908.981} C_VEL
LIN {X 0,Y 502.44,Z 604.933,A -85,B 0,C 180,E1 22907.577,E2 22907.577} C_VEL
LIN {X 0,Y 500.372,Z 589.833,A -85,B 0,C 180,E1 22906.167,E2 22906.167} C_VEL
LIN {X 0,Y 500.107,Z 570.371,A -85,B 0,C 180,E1 22904.516,E2 22904.516} C_VEL
LIN {X 0,Y 503.521,Z 523.336,A -85,B 0,C 180,E1 22900.791,E2 22900.791} C_VEL
LIN {X 0,Y 504.964,Z 505.176,A -85,B 0,C 180,E1 22899.317,E2 22899.317} C_VEL
LIN {X 0,Y 495.38,Z 485.22,A -85,B 0,C 180,E1 22896.359,E2 22896.359} C_VEL
LIN {X 0,Y 486.683,Z 467.82,A -85,B 0,C 180,E1 22893.548,E2 22893.548} C_VEL
LIN {X 0,Y 482.625,Z 459.634,A -85,B 0,C 180,E1 22892.17,E2 22892.17} C_VEL
LIN {X 0,Y 481.003,Z 456.245,A -85,B 0,C 180,E1 22891.589,E2 22891.589} C_VEL
LIN {X 0,Y 480.892,Z 455.576,A -85,B 0,C 180,E1 22891.458,E2 22891.458} C_VEL
LIN {X 0,Y 480.885,Z 455.586,A -85,B 0,C 180,E1 22887.893,E2 22887.893} C_VEL
LIN {X 0,Y 480.886,Z 455.585,A -85,B 0,C 180,E1 22884.31,E2 22884.31} C_VEL
LIN {X 0,Y 480.843,Z 455.59,A -85,B 0,C 180,E1 22880.656,E2 22880.656} C_VEL
LIN {X 0,Y 480.87,Z 455.587,A -85,B 0,C 180,E1 22876.923,E2 22876.923} C_VEL
LIN {X 0,Y 480.896,Z 455.586,A -85,B 0,C 180,E1 22873.336,E2 22873.336} C_VEL
LIN {X 0,Y 480.892,Z 455.585,A -85,B 0,C 180,E1 22869.575,E2 22869.575} C_VEL
LIN {X 0,Y 480.87,Z 455.587,A -85,B 0,C 180,E1 22865.967,E2 22865.967} C_VEL
LIN {X 0,Y 480.84,Z 455.589,A -85,B 0,C 180,E1 22862.264,E2 22862.264} C_VEL
LIN {X 0,Y 480.889,Z 455.583,A -85,B 0,C 180,E1 22858.689,E2 22858.689} C_VEL
LIN {X 0,Y 480.853,Z 455.587,A -85,B 0,C 180,E1 22855.229,E2 22855.229} C_VEL
LIN {X 0,Y 480.875,Z 455.573,A -85,B 0,C 180,E1 22851.751,E2 22851.751} C_VEL
LIN {X 0,Y 480.887,Z 455.581,A -85,B 0,C 180,E1 22848.243,E2 22848.243} C_VEL
LIN {X 0,Y 480.896,Z 455.584,A -85,B 0,C 180,E1 22844.566,E2 22844.566} C_VEL
LIN {X 0,Y 480.872,Z 455.582,A -85,B 0,C 180,E1 22840.947,E2 22840.947} C_VEL
LIN {X 0,Y 480.84,Z 455.578,A -85,B 0,C 180,E1 22837.246,E2 22837.246} C_VEL
LIN {X 0,Y 480.886,Z 455.581,A -85,B 0,C 180,E1 22833.653,E2 22833.653} C_VEL
LIN {X 0,Y 480.885,Z 455.585,A -85,B 0,C 180,E1 22830.065,E2 22830.065} C_VEL
LIN {X 0,Y 480.892,Z 455.583,A -85,B 0,C 180,E1 22826.423,E2 22826.423} C_VEL
LIN {X 0,Y 480.853,Z 455.586,A -85,B 0,C 180,E1 22822.786,E2 22822.786} C_VEL
LIN {X 0,Y 480.864,Z 455.58,A -85,B 0,C 180,E1 22819.082,E2 22819.082} C_VEL
LIN {X 0,Y 480.893,Z 455.585,A -85,B 0,C 180,E1 22815.491,E2 22815.491} C_VEL
LIN {X 0,Y 480.869,Z 455.586,A -85,B 0,C 180,E1 22811.87,E2 22811.87} C_VEL
LIN {X 0,Y 480.922,Z 455.802,A -85,B 0,C 180,E1 22809.713,E2 22809.713} C_VEL
LIN {X 0,Y 489.903,Z 478.537,A -85,B 0,C 180,E1 22806.768,E2 22806.768} C_VEL
LIN {X 0,Y 494.008,Z 490.369,A -85,B 0,C 180,E1 22805.369,E2 22805.369} C_VEL
LIN {X 0,Y 493.923,Z 497.806,A -85,B 0,C 180,E1 22804.806,E2 22804.806} C_VEL
LIN {X 0,Y 497.64,Z 518.494,A -85,B 0,C 180,E1 22804.15,E2 22804.15} C_VEL
LIN {X 0,Y 497.569,Z 522.676,A -85,B 0,C 180,E1 22804.084,E2 22804.084} C_VEL
LIN {X 0,Y 496.606,Z 530.37,A -85,B 0,C 180,E1 22804.027,E2 22804.027} C_VEL
LIN {X 0,Y 491.082,Z 550.878,A -85,B 0,C 180,E1 22804.111,E2 22804.111} C_VEL
LIN {X 0,Y 490.363,Z 557.478,A -85,B 0,C 180,E1 22804.053,E2 22804.053} C_VEL
LIN {X 0,Y 486.969,Z 758.2,A -85,B 0,C 180,E1 22800.832,E2 22800.832} C_VEL
LIN {X 0,Y 486.159,Z 779.107,A -85,B 0,C 180,E1 22800.291,E2 22800.291} C_VEL
LIN {X 0,Y 485.132,Z 798.636,A -85,B 0,C 180,E1 22799.571,E2 22799.571} C_VEL
LIN {X 0,Y 483.859,Z 817.821,A -85,B 0,C 180,E1 22798.646,E2 22798.646} C_VEL
LIN {X 0,Y 482.358,Z 837.027,A -85,B 0,C 180,E1 22797.478,E2 22797.478} C_VEL
LIN {X 0,Y 480.727,Z 855.456,A -85,B 0,C 180,E1 22796.097,E2 22796.097} C_VEL
LIN {X 0,Y 479.09,Z 872.608,A -85,B 0,C 180,E1 22794.538,E2 22794.538} C_VEL
LIN {X 0,Y 477.581,Z 887.777,A -85,B 0,C 180,E1 22792.9,E2 22792.9} C_VEL
LIN {X 0,Y 476.147,Z 902.384,A -85,B 0,C 180,E1 22791.043,E2 22791.043} C_VEL
LIN {X 0,Y 474.891,Z 915.773,A -85,B 0,C 180,E1 22789.03,E2 22789.03} C_VEL
LIN {X 0,Y 473.877,Z 927.578,A -85,B 0,C 180,E1 22786.928,E2 22786.928} C_VEL
LIN {X 0,Y 473.086,Z 938.077,A -85,B 0,C 180,E1 22784.691,E2 22784.691} C_VEL
LIN {X 0,Y 472.515,Z 947.087,A -85,B 0,C 180,E1 22782.34,E2 22782.34} C_VEL
LIN {X 0,Y 472.176,Z 954.279,A -85,B 0,C 180,E1 22779.999,E2 22779.999} C_VEL
LIN {X 0,Y 471.986,Z 960.405,A -85,B 0,C 180,E1 22777.424,E2 22777.424} C_VEL
LIN {X 0,Y 471.924,Z 964.549,A -85,B 0,C 180,E1 22774.983,E2 22774.983} C_VEL
LIN {X 0,Y 471.911,Z 967.076,A -85,B 0,C 180,E1 22772.549,E2 22772.549} C_VEL
LIN {X 0,Y 471.913,Z 967.976,A -85,B 0,C 180,E1 22770.121,E2 22770.121} C_VEL
LIN {X 0,Y 471.908,Z 967.261,A -85,B 0,C 180,E1 22767.692,E2 22767.692} C_VEL
LIN {X 0,Y 471.925,Z 964.983,A -85,B 0,C 180,E1 22765.26,E2 22765.26} C_VEL
LIN {X 0,Y 471.977,Z 961.09,A -85,B 0,C 180,E1 22762.819,E2 22762.819} C_VEL
LIN {X 0,Y 472.132,Z 955.545,A -85,B 0,C 180,E1 22760.368,E2 22760.368} C_VEL
LIN {X 0,Y 472.462,Z 948.167,A -85,B 0,C 180,E1 22757.883,E2 22757.883} C_VEL
LIN {X 0,Y 472.998,Z 939.232,A -85,B 0,C 180,E1 22755.502,E2 22755.502} C_VEL
LIN {X 0,Y 473.735,Z 929.242,A -85,B 0,C 180,E1 22753.319,E2 22753.319} C_VEL
LIN {X 0,Y 474.783,Z 916.943,A -85,B 0,C 180,E1 22751.075,E2 22751.075} C_VEL
LIN {X 0,Y 476.091,Z 903.003,A -85,B 0,C 180,E1 22748.953,E2 22748.953} C_VEL
LIN {X 0,Y 477.529,Z 888.378,A -85,B 0,C 180,E1 22747.079,E2 22747.079} C_VEL
LIN {X 0,Y 479.084,Z 872.688,A -85,B 0,C 180,E1 22745.379,E2 22745.379} C_VEL
LIN {X 0,Y 480.705,Z 855.718,A -85,B 0,C 180,E1 22743.834,E2 22743.834} C_VEL
LIN {X 0,Y 482.315,Z 837.498,A -85,B 0,C 180,E1 22742.464,E2 22742.464} C_VEL
LIN {X 0,Y 483.739,Z 819.268,A -85,B 0,C 180,E1 22741.345,E2 22741.345} C_VEL
LIN {X 0,Y 485.056,Z 799.916,A -85,B 0,C 180,E1 22740.395,E2 22740.395} C_VEL
LIN {X 0,Y 486.16,Z 779.096,A -85,B 0,C 180,E1 22739.619,E2 22739.619} C_VEL
LIN {X 0,Y 486.971,Z 758.137,A -85,B 0,C 180,E1 22739.077,E2 22739.077} C_VEL
LIN {X 0,Y 490.817,Z 526.537,A -85,B 0,C 180,E1 22735.353,E2 22735.353} C_VEL
LIN {X 0,Y 483.507,Z 499.789,A -85,B 0,C 180,E1 22734.249,E2 22734.249} C_VEL
LIN {X 0,Y 483.828,Z 490.522,A -85,B 0,C 180,E1 22733.107,E2 22733.107} C_VEL
LIN {X 0,Y 478.986,Z 474.498,A -85,B 0,C 180,E1 22730.455,E2 22730.455} C_VEL
LIN {X 0,Y 473.79,Z 459.33,A -85,B 0,C 180,E1 22727.794,E2 22727.794} C_VEL
LIN {X 0,Y 472.945,Z 456.576,A -85,B 0,C 180,E1 22727.315,E2 22727.315} C_VEL
LIN {X 0,Y 472.932,Z 456.571,A -85,B 0,C 180,E1 22723.692,E2 22723.692} C_VEL
LIN {X 0,Y 472.94,Z 456.573,A -85,B 0,C 180,E1 22719.994,E2 22719.994} C_VEL
LIN {X 0,Y 472.949,Z 456.576,A -85,B 0,C 180,E1 22716.343,E2 22716.343} C_VEL
LIN {X 0,Y 472.946,Z 456.584,A -85,B 0,C 180,E1 22715.064,E2 22715.064} C_VEL
LIN {X 0,Y 481.151,Z 479.346,A -85,B 0,C 180,E1 22711.719,E2 22711.719} C_VEL
LIN {X 0,Y 485.219,Z 491.907,A -85,B 0,C 180,E1 22709.981,E2 22709.981} C_VEL
LIN {X 0,Y 483.422,Z 523.79,A -85,B 0,C 180,E1 22706.668,E2 22706.668} C_VEL
LIN {X 0,Y 481.476,Z 559.928,A -85,B 0,C 180,E1 22702.98,E2 22702.98} C_VEL
LIN {X 0,Y 479.834,Z 595.361,A -85,B 0,C 180,E1 22699.412,E2 22699.412} C_VEL
LIN {X 0,Y 479.098,Z 614.071,A -85,B 0,C 180,E1 22697.582,E2 22697.582} C_VEL
LIN {X 0,Y 479.777,Z 620.014,A -85,B 0,C 180,E1 22697.43,E2 22697.43} C_VEL
LIN {X 0,Y 477.275,Z 756.668,A -85,B 0,C 180,E1 22694.905,E2 22694.905} C_VEL
LIN {X 0,Y 477.005,Z 773.699,A -85,B 0,C 180,E1 22694.351,E2 22694.351} C_VEL
LIN {X 0,Y 476.596,Z 788.484,A -85,B 0,C 180,E1 22693.652,E2 22693.652} C_VEL
LIN {X 0,Y 476.057,Z 803.572,A -85,B 0,C 180,E1 22692.7,E2 22692.7} C_VEL
LIN {X 0,Y 475.46,Z 817.32,A -85,B 0,C 180,E1 22691.586,E2 22691.586} C_VEL
LIN {X 0,Y 474.792,Z 830.944,A -85,B 0,C 180,E1 22690.189,E2 22690.189} C_VEL
LIN {X 0,Y 474.214,Z 842.262,A -85,B 0,C 180,E1 22688.732,E2 22688.732} C_VEL
LIN {X 0,Y 473.69,Z 852.826,A -85,B 0,C 180,E1 22687.032,E2 22687.032} C_VEL
LIN {X 0,Y 473.302,Z 861.108,A -85,B 0,C 180,E1 22685.334,E2 22685.334} C_VEL
LIN {X 0,Y 473.009,Z 868.387,A -85,B 0,C 180,E1 22683.393,E2 22683.393} C_VEL
LIN {X 0,Y 472.826,Z 873.564,A -85,B 0,C 180,E1 22681.454,E2 22681.454} C_VEL
LIN {X 0,Y 472.758,Z 876.954,A -85,B 0,C 180,E1 22679.515,E2 22679.515} C_VEL
LIN {X 0,Y 472.739,Z 878.599,A -85,B 0,C 180,E1 22677.576,E2 22677.576} C_VEL
LIN {X 0,Y 472.807,Z 878.524,A -85,B 0,C 180,E1 22675.513,E2 22675.513} C_VEL
LIN {X 0,Y 472.921,Z 876.677,A -85,B 0,C 180,E1 22673.562,E2 22673.562} C_VEL
LIN {X 0,Y 473.153,Z 873.107,A -85,B 0,C 180,E1 22671.616,E2 22671.616} C_VEL
LIN {X 0,Y 473.466,Z 867.946,A -85,B 0,C 180,E1 22669.77,E2 22669.77} C_VEL
LIN {X 0,Y 473.901,Z 860.97,A -85,B 0,C 180,E1 22667.944,E2 22667.944} C_VEL
LIN {X 0,Y 474.416,Z 852.865,A -85,B 0,C 180,E1 22666.311,E2 22666.311} C_VEL
LIN {X 0,Y 475.092,Z 842.221,A -85,B 0,C 180,E1 22664.623,E2 22664.623} C_VEL
LIN {X 0,Y 475.769,Z 830.958,A -85,B 0,C 180,E1 22663.214,E2 22663.214} C_VEL
LIN {X 0,Y 476.464,Z 818.029,A -85,B 0,C 180,E1 22661.921,E2 22661.921} C_VEL
LIN {X 0,Y 477.039,Z 804.293,A -85,B 0,C 180,E1 22660.852,E2 22660.852} C_VEL
LIN {X 0,Y 477.512,Z 789.581,A -85,B 0,C 180,E1 22659.964,E2 22659.964} C_VEL
LIN {X 0,Y 477.79,Z 773.778,A -85,B 0,C 180,E1 22659.281,E2 22659.281} C_VEL
LIN {X 0,Y 477.864,Z 758.071,A -85,B 0,C 180,E1 22658.831,E2 22658.831} C_VEL
LIN {X 0,Y 479.712,Z 695.249,A -85,B 0,C 180,E1 22657.433,E2 22657.433} C_VEL
LIN {X 0,Y 482.629,Z 633.113,A -85,B 0,C 180,E1 22655.946,E2 22655.946} C_VEL
LIN {X 0,Y 486.038,Z 624.106,A -85,B 0,C 180,E1 22655.187,E2 22655.187} C_VEL
LIN {X 0,Y 490.527,Z 593.364,A -85,B 0,C 180,E1 22651.512,E2 22651.512} C_VEL
LIN {X 0,Y 496.112,Z 566.932,A -85,B 0,C 180,E1 22648.128,E2 22648.128} C_VEL
LIN {X 0,Y 502.209,Z 546.529,A -85,B 0,C 180,E1 22645.292,E2 22645.292} C_VEL
LIN {X 0,Y 508.881,Z 531.066,A -85,B 0,C 180,E1 22642.914,E2 22642.914} C_VEL
LIN {X 0,Y 511.192,Z 526.737,A -85,B 0,C 180,E1 22642.109,E2 22642.109} C_VEL
LIN {X 0,Y 511.772,Z 525.324,A -85,B 0,C 180,E1 22640.907,E2 22640.907} C_VEL
LIN {X 0,Y 504.264,Z 537.282,A -85,B 0,C 180,E1 22639.414,E2 22639.414} C_VEL
LIN {X 0,Y 497.758,Z 551.923,A -85,B 0,C 180,E1 22637.751,E2 22637.751} C_VEL
LIN {X 0,Y 493.315,Z 567.176,A -85,B 0,C 180,E1 22636.119,E2 22636.119} C_VEL
LIN {X 0,Y 490.995,Z 583.664,A -85,B 0,C 180,E1 22634.376,E2 22634.376} C_VEL
LIN {X 0,Y 491.195,Z 598.067,A -85,B 0,C 180,E1 22632.835,E2 22632.835} C_VEL
LIN {X 0,Y 493.627,Z 611.777,A -85,B 0,C 180,E1 22631.325,E2 22631.325} C_VEL
LIN {X 0,Y 498.053,Z 624.121,A -85,B 0,C 180,E1 22629.926,E2 22629.926} C_VEL
LIN {X 0,Y 504.305,Z 635.157,A -85,B 0,C 180,E1 22628.633,E2 22628.633} C_VEL
LIN {X 0,Y 511.736,Z 644.521,A -85,B 0,C 180,E1 22627.509,E2 22627.509} C_VEL
LIN {X 0,Y 521.54,Z 653.733,A -85,B 0,C 180,E1 22626.371,E2 22626.371} C_VEL
LIN {X 0,Y 533.121,Z 661.859,A -85,B 0,C 180,E1 22625.33,E2 22625.33} C_VEL
LIN {X 0,Y 536.354,Z 663.989,A -85,B 0,C 180,E1 22625.066,E2 22625.066} C_VEL
LIN {X 0,Y 526.671,Z 680.346,A -85,B 0,C 180,E1 22624.454,E2 22624.454} C_VEL
LIN {X 0,Y 523.677,Z 685.832,A -85,B 0,C 180,E1 22624.236,E2 22624.236} C_VEL
LIN {X 0,Y 510.675,Z 704.682,A -85,B 0,C 180,E1 22623.581,E2 22623.581} C_VEL
LIN {X 0,Y 501.846,Z 720.097,A -85,B 0,C 180,E1 22622.951,E2 22622.951} C_VEL
LIN {X 0,Y 495.405,Z 734.659,A -85,B 0,C 180,E1 22622.265,E2 22622.265} C_VEL
LIN {X 0,Y 488.408,Z 752.963,A -85,B 0,C 180,E1 22621.366,E2 22621.366} C_VEL
LIN {X 0,Y 486.35,Z 773.429,A -85,B 0,C 180,E1 22621.167,E2 22621.167} C_VEL
LIN {X 0,Y 485.678,Z 806.498,A -85,B 0,C 180,E1 22620.602,E2 22620.602} C_VEL
LIN {X 0,Y 484.787,Z 827.046,A -85,B 0,C 180,E1 22620.045,E2 22620.045} C_VEL
LIN {X 0,Y 483.623,Z 847.538,A -85,B 0,C 180,E1 22619.255,E2 22619.255} C_VEL
LIN {X 0,Y 482.301,Z 866.934,A -85,B 0,C 180,E1 22618.276,E2 22618.276} C_VEL
LIN {X 0,Y 480.847,Z 885.776,A -85,B 0,C 180,E1 22617.09,E2 22617.09} C_VEL
LIN {X 0,Y 479.287,Z 904.524,A -85,B 0,C 180,E1 22615.651,E2 22615.651} C_VEL
LIN {X 0,Y 477.767,Z 922.1,A -85,B 0,C 180,E1 22614.025,E2 22614.025} C_VEL
LIN {X 0,Y 476.41,Z 938.231,A -85,B 0,C 180,E1 22612.25,E2 22612.25} C_VEL
LIN {X 0,Y 475.148,Z 953.129,A -85,B 0,C 180,E1 22610.318,E2 22610.318} C_VEL
LIN {X 0,Y 473.835,Z 971.87,A -85,B 0,C 180,E1 22607.437,E2 22607.437} C_VEL
LIN {X 0,Y 473.208,Z 982.341,A -85,B 0,C 180,E1 22605.529,E2 22605.529} C_VEL
LIN {X 0,Y 472.732,Z 990.941,A -85,B 0,C 180,E1 22603.704,E2 22603.704} C_VEL
LIN {X 0,Y 472.337,Z 999.71,A -85,B 0,C 180,E1 22601.478,E2 22601.478} C_VEL
LIN {X 0,Y 472.107,Z 1005.94,A -85,B 0,C 180,E1 22599.386,E2 22599.386} C_VEL
LIN {X 0,Y 471.978,Z 1010.716,A -85,B 0,C 180,E1 22597.303,E2 22597.303} C_VEL
LIN {X 0,Y 471.926,Z 1014.803,A -85,B 0,C 180,E1 22594.862,E2 22594.862} C_VEL
LIN {X 0,Y 471.908,Z 1017.045,A -85,B 0,C 180,E1 22592.551,E2 22592.551} C_VEL
LIN {X 0,Y 471.905,Z 1017.957,A -85,B 0,C 180,E1 22590.243,E2 22590.243} C_VEL
LIN {X 0,Y 471.909,Z 1017.21,A -85,B 0,C 180,E1 22587.694,E2 22587.694} C_VEL
LIN {X 0,Y 471.922,Z 1015.211,A -85,B 0,C 180,E1 22585.505,E2 22585.505} C_VEL
LIN {X 0,Y 471.974,Z 1011.227,A -85,B 0,C 180,E1 22582.943,E2 22582.943} C_VEL
LIN {X 0,Y 472.096,Z 1006.238,A -85,B 0,C 180,E1 22580.732,E2 22580.732} C_VEL
LIN {X 0,Y 472.286,Z 1000.89,A -85,B 0,C 180,E1 22578.893,E2 22578.893} C_VEL
LIN {X 0,Y 472.68,Z 992.165,A -85,B 0,C 180,E1 22576.546,E2 22576.546} C_VEL
LIN {X 0,Y 473.197,Z 982.706,A -85,B 0,C 180,E1 22574.476,E2 22574.476} C_VEL
LIN {X 0,Y 473.93,Z 971.063,A -85,B 0,C 180,E1 22572.315,E2 22572.315} C_VEL
LIN {X 0,Y 474.834,Z 958.081,A -85,B 0,C 180,E1 22570.312,E2 22570.312} C_VEL
LIN {X 0,Y 475.945,Z 943.457,A -85,B 0,C 180,E1 22568.366,E2 22568.366} C_VEL
LIN {X 0,Y 477.452,Z 925.237,A -85,B 0,C 180,E1 22566.293,E2 22566.293} C_VEL
LIN {X 0,Y 478.953,Z 908.252,A -85,B 0,C 180,E1 22564.663,E2 22564.663} C_VEL
LIN {X 0,Y 480.417,Z 890.456,A -85,B 0,C 180,E1 22563.233,E2 22563.233} C_VEL
LIN {X 0,Y 481.925,Z 871.288,A -85,B 0,C 180,E1 22561.971,E2 22561.971} C_VEL
LIN {X 0,Y 483.261,Z 852.167,A -85,B 0,C 180,E1 22560.958,E2 22560.958} C_VEL
LIN {X 0,Y 484.443,Z 831.985,A -85,B 0,C 180,E1 22560.125,E2 22560.125} C_VEL
LIN {X 0,Y 485.446,Z 810.709,A -85,B 0,C 180,E1 22559.494,E2 22559.494} C_VEL
LIN {X 0,Y 486.055,Z 787.671,A -85,B 0,C 180,E1 22559.052,E2 22559.052} C_VEL
LIN {X 0,Y 486.703,Z 766.379,A -85,B 0,C 180,E1 22558.739,E2 22558.739} C_VEL
LIN {X 0,Y 492.562,Z 748.575,A -85,B 0,C 180,E1 22557.802,E2 22557.802} C_VEL
LIN {X 0,Y 497.855,Z 735.371,A -85,B 0,C 180,E1 22557.164,E2 22557.164} C_VEL
LIN {X 0,Y 504.614,Z 720.539,A -85,B 0,C 180,E1 22556.508,E2 22556.508} C_VEL
LIN {X 0,Y 513.911,Z 704.293,A -85,B 0,C 180,E1 22555.922,E2 22555.922} C_VEL
LIN {X 0,Y 526.166,Z 685.763,A -85,B 0,C 180,E1 22555.377,E2 22555.377} C_VEL
LIN {X 0,Y 534.598,Z 670.277,A -85,B 0,C 180,E1 22554.827,E2 22554.827} C_VEL
LIN {X 0,Y 537.457,Z 665.164,A -85,B 0,C 180,E1 22554.654,E2 22554.654} C_VEL
LIN {X 0,Y 526.362,Z 658.349,A -85,B 0,C 180,E1 22553.467,E2 22553.467} C_VEL
LIN {X 0,Y 517.159,Z 650.475,A -85,B 0,C 180,E1 22552.255,E2 22552.255} C_VEL
LIN {X 0,Y 509.46,Z 641.381,A -85,B 0,C 180,E1 22551.003,E2 22551.003} C_VEL
LIN {X 0,Y 502.779,Z 630.098,A -85,B 0,C 180,E1 22549.61,E2 22549.61} C_VEL
LIN {X 0,Y 498.004,Z 617.65,A -85,B 0,C 180,E1 22548.225,E2 22548.225} C_VEL
LIN {X 0,Y 494.768,Z 603.079,A -85,B 0,C 180,E1 22546.759,E2 22546.759} C_VEL
LIN {X 0,Y 493.348,Z 586.78,A -85,B 0,C 180,E1 22545.271,E2 22545.271} C_VEL
LIN {X 0,Y 493.851,Z 565.545,A -85,B 0,C 180,E1 22543.501,E2 22543.501} C_VEL
LIN {X 0,Y 497.088,Z 525.879,A -85,B 0,C 180,E1 22540.331,E2 22540.331} C_VEL
LIN {X 0,Y 498.495,Z 509.119,A -85,B 0,C 180,E1 22538.962,E2 22538.962} C_VEL
LIN {X 0,Y 489.225,Z 489.83,A -85,B 0,C 180,E1 22536.058,E2 22536.058} C_VEL
LIN {X 0,Y 480.796,Z 472.863,A -85,B 0,C 180,E1 22533.299,E2 22533.299} C_VEL
LIN {X 0,Y 476.731,Z 464.77,A -85,B 0,C 180,E1 22531.906,E2 22531.906} C_VEL
LIN {X 0,Y 474.747,Z 460.712,A -85,B 0,C 180,E1 22531.204,E2 22531.204} C_VEL
LIN {X 0,Y 473.09,Z 457.466,A -85,B 0,C 180,E1 22530.62,E2 22530.62} C_VEL
LIN {X 0,Y 472.929,Z 456.576,A -85,B 0,C 180,E1 22530.491,E2 22530.491} C_VEL
LIN {X 0,Y 472.917,Z 456.578,A -85,B 0,C 180,E1 22526.765,E2 22526.765} C_VEL
LIN {X 0,Y 472.953,Z 456.573,A -85,B 0,C 180,E1 22523.131,E2 22523.131} C_VEL
LIN {X 0,Y 472.934,Z 456.577,A -85,B 0,C 180,E1 22519.514,E2 22519.514} C_VEL
LIN {X 0,Y 472.949,Z 456.575,A -85,B 0,C 180,E1 22515.952,E2 22515.952} C_VEL
LIN {X 0,Y 472.903,Z 456.58,A -85,B 0,C 180,E1 22512.33,E2 22512.33} C_VEL
LIN {X 0,Y 472.931,Z 456.575,A -85,B 0,C 180,E1 22508.633,E2 22508.633} C_VEL
LIN {X 0,Y 472.954,Z 456.573,A -85,B 0,C 180,E1 22504.972,E2 22504.972} C_VEL
LIN {X 0,Y 472.956,Z 456.57,A -85,B 0,C 180,E1 22501.09,E2 22501.09} C_VEL
LIN {X 0,Y 472.93,Z 456.574,A -85,B 0,C 180,E1 22497.455,E2 22497.455} C_VEL
LIN {X 0,Y 472.908,Z 456.576,A -85,B 0,C 180,E1 22493.688,E2 22493.688} C_VEL
LIN {X 0,Y 472.948,Z 456.571,A -85,B 0,C 180,E1 22490.117,E2 22490.117} C_VEL
LIN {X 0,Y 472.941,Z 456.563,A -85,B 0,C 180,E1 22486.529,E2 22486.529} C_VEL
LIN {X 0,Y 472.95,Z 456.565,A -85,B 0,C 180,E1 22482.911,E2 22482.911} C_VEL
